LIN {X 0,Y 236.637,Z 407.423,A -85,B 0,C 180,E1 -20816.053,E2 -20816.053} C_VEL
LIN {X 0,Y 232.607,Z 398.672,A -85,B 0,C 180,E1 -20818.068,E2 -20818.068} C_VEL
LIN {X 0,Y 229.513,Z 389.934,A -85,B 0,C 180,E1 -20819.777,E2 -20819.777} C_VEL
LIN {X 0,Y 225.786,Z 379.77,A -85,B 0,C 180,E1 -20821.562,E2 -20821.562} C_VEL
LIN {X 0,Y 220.741,Z 368.882,A -85,B 0,C 180,E1 -20823.411,E2 -20823.411} C_VEL
LIN {X 0,Y 216.833,Z 361.674,A -85,B 0,C 180,E1 -20824.638,E2 -20824.638} C_VEL
LIN {X 0,Y 215.315,Z 358.971,A -85,B 0,C 180,E1 -20825.078,E2 -20825.078} C_VEL
LIN {X 0,Y 213.899,Z 356.173,A -85,B 0,C 180,E1 -20825.487,E2 -20825.487} C_VEL
LIN {X 0,Y 213.743,Z 355.361,A -85,B 0,C 180,E1 -20825.592,E2 -20825.592} C_VEL
LIN {X 0,Y 213.776,Z 355.356,A -85,B 0,C 180,E1 -20828.655,E2 -20828.655} C_VEL
LIN {X 0,Y 213.806,Z 355.353,A -85,B 0,C 180,E1 -20833.686,E2 -20833.686} C_VEL
LIN {X 0,Y 213.809,Z 355.352,A -85,B 0,C 180,E1 -20836.349,E2 -20836.349} C_VEL
LIN {X 0,Y 213.792,Z 355.354,A -85,B 0,C 180,E1 -20839.119,E2 -20839.119} C_VEL
LIN {X 0,Y 213.752,Z 355.359,A -85,B 0,C 180,E1 -20843.715,E2 -20843.715} C_VEL
LIN {X 0,Y 213.794,Z 355.352,A -85,B 0,C 180,E1 -20848.725,E2 -20848.725} C_VEL
LIN {X 0,Y 213.824,Z 355.349,A -85,B 0,C 180,E1 -20852.604,E2 -20852.604} C_VEL
LIN {X 0,Y 213.818,Z 355.35,A -85,B 0,C 180,E1 -20856.975,E2 -20856.975} C_VEL
LIN {X 0,Y 213.943,Z 355.336,A -85,B 0,C 180,E1 -20862.805,E2 -20862.805} C_VEL
LIN {X 0,Y 213.98,Z 355.328,A -85,B 0,C 180,E1 -20866.709,E2 -20866.709} C_VEL
LIN {X 0,Y 214.166,Z 355.301,A -85,B 0,C 180,E1 -20870.557,E2 -20870.557} C_VEL
LIN {X 0,Y 214.226,Z 355.299,A -85,B 0,C 180,E1 -20872.461,E2 -20872.461} C_VEL
LIN {X 0,Y 214.445,Z 355.244,A -85,B 0,C 180,E1 -20878.123,E2 -20878.123} C_VEL
LIN {X 0,Y 214.546,Z 355.244,A -85,B 0,C 180,E1 -20880.001,E2 -20880.001} C_VEL
LIN {X 0,Y 214.446,Z 355.269,A -85,B 0,C 180,E1 -20881.879,E2 -20881.879} C_VEL
LIN {X 0,Y 214.227,Z 355.3,A -85,B 0,C 180,E1 -20887.541,E2 -20887.541} C_VEL
LIN {X 0,Y 214.022,Z 355.327,A -85,B 0,C 180,E1 -20891.364,E2 -20891.364} C_VEL
LIN {X 0,Y 213.913,Z 355.341,A -85,B 0,C 180,E1 -20895.239,E2 -20895.239} C_VEL
LIN {X 0,Y 213.82,Z 355.351,A -85,B 0,C 180,E1 -20899.19,E2 -20899.19} C_VEL
LIN {X 0,Y 213.812,Z 355.353,A -85,B 0,C 180,E1 -20903.232,E2 -20903.232} C_VEL
LIN {X 0,Y 213.831,Z 355.54,A -85,B 0,C 180,E1 -20907.451,E2 -20907.451} C_VEL
LIN {X 0,Y 214.005,Z 357.167,A -85,B 0,C 180,E1 -20911.699,E2 -20911.699} C_VEL
LIN {X 0,Y 214.27,Z 359.11,A -85,B 0,C 180,E1 -20916.186,E2 -20916.186} C_VEL
LIN {X 0,Y 214.638,Z 361.528,A -85,B 0,C 180,E1 -20921.141,E2 -20921.141} C_VEL
LIN {X 0,Y 214.75,Z 363.018,A -85,B 0,C 180,E1 -20923.947,E2 -20923.947} C_VEL
LIN {X 0,Y 214.71,Z 364.508,A -85,B 0,C 180,E1 -20926.577,E2 -20926.577} C_VEL
LIN {X 0,Y 214.484,Z 365.996,A -85,B 0,C 180,E1 -20929.055,E2 -20929.055} C_VEL
LIN {X 0,Y 214.063,Z 367.842,A -85,B 0,C 180,E1 -20931.996,E2 -20931.996} C_VEL
LIN {X 0,Y 213.615,Z 369.611,A -85,B 0,C 180,E1 -20934.67,E2 -20934.67} C_VEL
LIN {X 0,Y 214.471,Z 372.783,A -85,B 0,C 180,E1 -20935.009,E2 -20935.009} C_VEL
LIN {X 0,Y 218.045,Z 383.16,A -85,B 0,C 180,E1 -20936.461,E2 -20936.461} C_VEL
LIN {X 0,Y 221.063,Z 395.512,A -85,B 0,C 180,E1 -20938.295,E2 -20938.295} C_VEL
LIN {X 0,Y 222.714,Z 405.325,A -85,B 0,C 180,E1 -20939.887,E2 -20939.887} C_VEL
LIN {X 0,Y 223.669,Z 414.982,A -85,B 0,C 180,E1 -20941.62,E2 -20941.62} C_VEL
LIN {X 0,Y 223.891,Z 424.106,A -85,B 0,C 180,E1 -20943.447,E2 -20943.447} C_VEL
LIN {X 0,Y 223.651,Z 428.588,A -85,B 0,C 180,E1 -20944.401,E2 -20944.401} C_VEL
LIN {X 0,Y 220.94,Z 438.166,A -85,B 0,C 180,E1 -20946.571,E2 -20946.571} C_VEL
LIN {X 0,Y 218.739,Z 445.725,A -85,B 0,C 180,E1 -20948.713,E2 -20948.713} C_VEL
LIN {X 0,Y 216.763,Z 452.535,A -85,B 0,C 180,E1 -20951.081,E2 -20951.081} C_VEL
LIN {X 0,Y 215.226,Z 457.725,A -85,B 0,C 180,E1 -20953.259,E2 -20953.259} C_VEL
LIN {X 0,Y 213.717,Z 460.581,A -85,B 0,C 180,E1 -20954.599,E2 -20954.599} C_VEL
LIN {X 0,Y 209.734,Z 464.564,A -85,B 0,C 180,E1 -20956.799,E2 -20956.799} C_VEL
LIN {X 0,Y 206.003,Z 467.926,A -85,B 0,C 180,E1 -20959.155,E2 -20959.155} C_VEL
LIN {X 0,Y 204.917,Z 469.562,A -85,B 0,C 180,E1 -20960.709,E2 -20960.709} C_VEL
LIN {X 0,Y 204.405,Z 472.228,A -85,B 0,C 180,E1 -20964.08,E2 -20964.08} C_VEL
LIN {X 0,Y 204.339,Z 473.292,A -85,B 0,C 180,E1 -20966.056,E2 -20966.056} C_VEL
LIN {X 0,Y 204.335,Z 473.885,A -85,B 0,C 180,E1 -20968.029,E2 -20968.029} C_VEL
LIN {X 0,Y 204.443,Z 474.044,A -85,B 0,C 180,E1 -20970,E2 -20970} C_VEL
LIN {X 0,Y 204.334,Z 473.885,A -85,B 0,C 180,E1 -20971.971,E2 -20971.971} C_VEL
LIN {X 0,Y 204.299,Z 473.291,A -85,B 0,C 180,E1 -20973.945,E2 -20973.945} C_VEL
LIN {X 0,Y 204.643,Z 470.836,A -85,B 0,C 180,E1 -20977.896,E2 -20977.896} C_VEL
LIN {X 0,Y 205.316,Z 467.882,A -85,B 0,C 180,E1 -20980.852,E2 -20980.852} C_VEL
LIN {X 0,Y 206.328,Z 463.887,A -85,B 0,C 180,E1 -20983.794,E2 -20983.794} C_VEL
LIN {X 0,Y 207.985,Z 458.757,A -85,B 0,C 180,E1 -20986.692,E2 -20986.692} C_VEL
LIN {X 0,Y 209.651,Z 453.494,A -85,B 0,C 180,E1 -20989.077,E2 -20989.077} C_VEL
LIN {X 0,Y 211.297,Z 448.555,A -85,B 0,C 180,E1 -20990.95,E2 -20990.95} C_VEL
LIN {X 0,Y 212.934,Z 442.852,A -85,B 0,C 180,E1 -20992.818,E2 -20992.818} C_VEL
LIN {X 0,Y 215.477,Z 434.299,A -85,B 0,C 180,E1 -20995.088,E2 -20995.088} C_VEL
LIN {X 0,Y 217.129,Z 428.388,A -85,B 0,C 180,E1 -20996.427,E2 -20996.427} C_VEL
LIN {X 0,Y 217.265,Z 418.838,A -85,B 0,C 180,E1 -20998.508,E2 -20998.508} C_VEL
LIN {X 0,Y 216.618,Z 409.561,A -85,B 0,C 180,E1 -21000.324,E2 -21000.324} C_VEL
LIN {X 0,Y 215.169,Z 399.419,A -85,B 0,C 180,E1 -21002.119,E2 -21002.119} C_VEL
LIN {X 0,Y 213.245,Z 390.302,A -85,B 0,C 180,E1 -21003.61,E2 -21003.61} C_VEL
LIN {X 0,Y 210.499,Z 380.51,A -85,B 0,C 180,E1 -21005.113,E2 -21005.113} C_VEL
LIN {X 0,Y 207.569,Z 372.479,A -85,B 0,C 180,E1 -21006.34,E2 -21006.34} C_VEL
LIN {X 0,Y 206.759,Z 369.447,A -85,B 0,C 180,E1 -21006.724,E2 -21006.724} C_VEL
LIN {X 0,Y 207.256,Z 367.276,A -85,B 0,C 180,E1 -21010.112,E2 -21010.112} C_VEL
LIN {X 0,Y 207.547,Z 365.774,A -85,B 0,C 180,E1 -21012.628,E2 -21012.628} C_VEL
LIN {X 0,Y 207.694,Z 364.302,A -85,B 0,C 180,E1 -21015.284,E2 -21015.284} C_VEL
LIN {X 0,Y 207.502,Z 361.92,A -85,B 0,C 180,E1 -21019.944,E2 -21019.944} C_VEL
LIN {X 0,Y 207.201,Z 359.698,A -85,B 0,C 180,E1 -21024.786,E2 -21024.786} C_VEL
LIN {X 0,Y 206.933,Z 357.824,A -85,B 0,C 180,E1 -21029.372,E2 -21029.372} C_VEL
LIN {X 0,Y 206.733,Z 356.236,A -85,B 0,C 180,E1 -21033.771,E2 -21033.771} C_VEL
LIN {X 0,Y 206.737,Z 356.236,A -85,B 0,C 180,E1 -21038.04,E2 -21038.04} C_VEL
LIN {X 0,Y 206.869,Z 356.218,A -85,B 0,C 180,E1 -21042.195,E2 -21042.195} C_VEL
LIN {X 0,Y 206.886,Z 356.214,A -85,B 0,C 180,E1 -21046.243,E2 -21046.243} C_VEL
LIN {X 0,Y 207.106,Z 356.186,A -85,B 0,C 180,E1 -21050.23,E2 -21050.23} C_VEL
LIN {X 0,Y 207.168,Z 356.179,A -85,B 0,C 180,E1 -21052.2,E2 -21052.2} C_VEL
LIN {X 0,Y 207.382,Z 356.149,A -85,B 0,C 180,E1 -21058.057,E2 -21058.057} C_VEL
LIN {X 0,Y 207.512,Z 356.118,A -85,B 0,C 180,E1 -21059.999,E2 -21059.999} C_VEL
LIN {X 0,Y 207.382,Z 356.122,A -85,B 0,C 180,E1 -21061.941,E2 -21061.941} C_VEL
LIN {X 0,Y 207.167,Z 356.178,A -85,B 0,C 180,E1 -21067.798,E2 -21067.798} C_VEL
LIN {X 0,Y 206.981,Z 356.202,A -85,B 0,C 180,E1 -21071.754,E2 -21071.754} C_VEL
LIN {X 0,Y 206.866,Z 356.213,A -85,B 0,C 180,E1 -21075.77,E2 -21075.77} C_VEL
LIN {X 0,Y 206.762,Z 356.222,A -85,B 0,C 180,E1 -21079.87,E2 -21079.87} C_VEL
LIN {X 0,Y 206.745,Z 356.228,A -85,B 0,C 180,E1 -21084.073,E2 -21084.073} C_VEL
LIN {X 0,Y 206.742,Z 356.232,A -85,B 0,C 180,E1 -21088.418,E2 -21088.418} C_VEL
LIN {X 0,Y 206.707,Z 356.235,A -85,B 0,C 180,E1 -21092.955,E2 -21092.955} C_VEL
LIN {X 0,Y 206.723,Z 356.235,A -85,B 0,C 180,E1 -21097.729,E2 -21097.729} C_VEL
LIN {X 0,Y 206.721,Z 356.235,A -85,B 0,C 180,E1 -21101.588,E2 -21101.588} C_VEL
LIN {X 0,Y 206.715,Z 356.234,A -85,B 0,C 180,E1 -21105.557,E2 -21105.557} C_VEL
LIN {X 0,Y 206.717,Z 356.235,A -85,B 0,C 180,E1 -21109.762,E2 -21109.762} C_VEL
LIN {X 0,Y 206.724,Z 356.235,A -85,B 0,C 180,E1 -21113.053,E2 -21113.053} C_VEL
LIN {X 0,Y 207.763,Z 359.167,A -85,B 0,C 180,E1 -21113.467,E2 -21113.467} C_VEL
LIN {X 0,Y 209.141,Z 361.156,A -85,B 0,C 180,E1 -21113.859,E2 -21113.859} C_VEL
LIN {X 0,Y 214.594,Z 371.285,A -85,B 0,C 180,E1 -21115.68,E2 -21115.68} C_VEL
LIN {X 0,Y 219.935,Z 383.191,A -85,B 0,C 180,E1 -21117.855,E2 -21117.855} C_VEL
LIN {X 0,Y 223.964,Z 394.74,A -85,B 0,C 180,E1 -21120.075,E2 -21120.075} C_VEL
LIN {X 0,Y 226.905,Z 403.215,A -85,B 0,C 180,E1 -21121.899,E2 -21121.899} C_VEL
LIN {X 0,Y 230.392,Z 410.806,A -85,B 0,C 180,E1 -21123.814,E2 -21123.814} C_VEL
LIN {X 0,Y 235.845,Z 419.628,A -85,B 0,C 180,E1 -21126.391,E2 -21126.391} C_VEL
LIN {X 0,Y 242.561,Z 427.895,A -85,B 0,C 180,E1 -21129.18,E2 -21129.18} C_VEL
LIN {X 0,Y 250.879,Z 435.889,A -85,B 0,C 180,E1 -21132.259,E2 -21132.259} C_VEL
LIN {X 0,Y 258.448,Z 441.903,A -85,B 0,C 180,E1 -21134.867,E2 -21134.867} C_VEL
LIN {X 0,Y 267.451,Z 447.962,A -85,B 0,C 180,E1 -21137.865,E2 -21137.865} C_VEL
LIN {X 0,Y 274.648,Z 452.392,A -85,B 0,C 180,E1 -21140.426,E2 -21140.426} C_VEL
LIN {X 0,Y 280.647,Z 455.777,A -85,B 0,C 180,E1 -21142.807,E2 -21142.807} C_VEL
LIN {X 0,Y 283.645,Z 457.491,A -85,B 0,C 180,E1 -21144.312,E2 -21144.312} C_VEL
LIN {X 0,Y 285.802,Z 458.811,A -85,B 0,C 180,E1 -21145.769,E2 -21145.769} C_VEL
LIN {X 0,Y 288.397,Z 459.95,A -85,B 0,C 180,E1 -21147.597,E2 -21147.597} C_VEL
LIN {X 0,Y 289.483,Z 460.298,A -85,B 0,C 180,E1 -21148.609,E2 -21148.609} C_VEL
LIN {X 0,Y 290.505,Z 460.469,A -85,B 0,C 180,E1 -21150,E2 -21150} C_VEL
LIN {X 0,Y 289.451,Z 460.299,A -85,B 0,C 180,E1 -21151.391,E2 -21151.391} C_VEL
LIN {X 0,Y 287.782,Z 459.753,A -85,B 0,C 180,E1 -21152.8,E2 -21152.8} C_VEL
LIN {X 0,Y 285.767,Z 458.812,A -85,B 0,C 180,E1 -21154.231,E2 -21154.231} C_VEL
LIN {X 0,Y 282.769,Z 456.952,A -85,B 0,C 180,E1 -21156.199,E2 -21156.199} C_VEL
LIN {X 0,Y 280.618,Z 455.778,A -85,B 0,C 180,E1 -21157.194,E2 -21157.194} C_VEL
LIN {X 0,Y 274.681,Z 452.391,A -85,B 0,C 180,E1 -21159.573,E2 -21159.573} C_VEL
LIN {X 0,Y 267.469,Z 447.961,A -85,B 0,C 180,E1 -21162.134,E2 -21162.134} C_VEL
LIN {X 0,Y 258.46,Z 441.872,A -85,B 0,C 180,E1 -21165.143,E2 -21165.143} C_VEL
LIN {X 0,Y 250.162,Z 435.246,A -85,B 0,C 180,E1 -21168.001,E2 -21168.001} C_VEL
LIN {X 0,Y 242.538,Z 427.896,A -85,B 0,C 180,E1 -21170.822,E2 -21170.822} C_VEL
LIN {X 0,Y 235.837,Z 419.654,A -85,B 0,C 180,E1 -21173.604,E2 -21173.604} C_VEL
LIN {X 0,Y 230.413,Z 410.784,A -85,B 0,C 180,E1 -21176.188,E2 -21176.188} C_VEL
LIN {X 0,Y 226.497,Z 402.035,A -85,B 0,C 180,E1 -21178.37,E2 -21178.37} C_VEL
LIN {X 0,Y 222.706,Z 390.823,A -85,B 0,C 180,E1 -21180.693,E2 -21180.693} C_VEL
LIN {X 0,Y 219.275,Z 381.514,A -85,B 0,C 180,E1 -21182.446,E2 -21182.446} C_VEL
LIN {X 0,Y 214.031,Z 370.166,A -85,B 0,C 180,E1 -21184.516,E2 -21184.516} C_VEL
LIN {X 0,Y 208.531,Z 360.174,A -85,B 0,C 180,E1 -21186.339,E2 -21186.339} C_VEL
LIN {X 0,Y 207.1,Z 357.827,A -85,B 0,C 180,E1 -21186.767,E2 -21186.767} C_VEL
LIN {X 0,Y 206.708,Z 356.237,A -85,B 0,C 180,E1 -21186.941,E2 -21186.941} C_VEL
LIN {X 0,Y 206.716,Z 356.236,A -85,B 0,C 180,E1 -21191.588,E2 -21191.588} C_VEL
LIN {X 0,Y 206.715,Z 356.235,A -85,B 0,C 180,E1 -21195.558,E2 -21195.558} C_VEL
LIN {X 0,Y 206.722,Z 356.234,A -85,B 0,C 180,E1 -21199.765,E2 -21199.765} C_VEL
LIN {X 0,Y 206.723,Z 356.235,A -85,B 0,C 180,E1 -21202.271,E2 -21202.271} C_VEL
LIN {X 0,Y 206.707,Z 356.235,A -85,B 0,C 180,E1 -21207.045,E2 -21207.045} C_VEL
LIN {X 0,Y 206.765,Z 356.229,A -85,B 0,C 180,E1 -21212.097,E2 -21212.097} C_VEL
LIN {X 0,Y 206.753,Z 356.229,A -85,B 0,C 180,E1 -21216.605,E2 -21216.605} C_VEL
LIN {X 0,Y 206.872,Z 356.215,A -85,B 0,C 180,E1 -21222.198,E2 -21222.198} C_VEL
LIN {X 0,Y 206.913,Z 356.207,A -85,B 0,C 180,E1 -21226.247,E2 -21226.247} C_VEL
LIN {X 0,Y 207.105,Z 356.18,A -85,B 0,C 180,E1 -21230.232,E2 -21230.232} C_VEL
LIN {X 0,Y 207.167,Z 356.178,A -85,B 0,C 180,E1 -21232.202,E2 -21232.202} C_VEL
LIN {X 0,Y 207.382,Z 356.122,A -85,B 0,C 180,E1 -21238.059,E2 -21238.059} C_VEL
LIN {X 0,Y 207.512,Z 356.118,A -85,B 0,C 180,E1 -21240.001,E2 -21240.001} C_VEL
LIN {X 0,Y 207.382,Z 356.149,A -85,B 0,C 180,E1 -21241.943,E2 -21241.943} C_VEL
LIN {X 0,Y 207.168,Z 356.179,A -85,B 0,C 180,E1 -21247.8,E2 -21247.8} C_VEL
LIN {X 0,Y 206.941,Z 356.209,A -85,B 0,C 180,E1 -21251.758,E2 -21251.758} C_VEL
LIN {X 0,Y 206.846,Z 356.221,A -85,B 0,C 180,E1 -21255.773,E2 -21255.773} C_VEL
LIN {X 0,Y 206.858,Z 356.22,A -85,B 0,C 180,E1 -21257.955,E2 -21257.955} C_VEL
LIN {X 0,Y 206.755,Z 356.233,A -85,B 0,C 180,E1 -21263.397,E2 -21263.397} C_VEL
LIN {X 0,Y 206.732,Z 356.236,A -85,B 0,C 180,E1 -21266.229,E2 -21266.229} C_VEL
LIN {X 0,Y 206.933,Z 357.826,A -85,B 0,C 180,E1 -21270.628,E2 -21270.628} C_VEL
LIN {X 0,Y 207.209,Z 359.819,A -85,B 0,C 180,E1 -21275.51,E2 -21275.51} C_VEL
LIN {X 0,Y 207.507,Z 361.919,A -85,B 0,C 180,E1 -21280.055,E2 -21280.055} C_VEL
LIN {X 0,Y 207.633,Z 363.198,A -85,B 0,C 180,E1 -21282.608,E2 -21282.608} C_VEL
LIN {X 0,Y 207.679,Z 364.638,A -85,B 0,C 180,E1 -21285.29,E2 -21285.29} C_VEL
LIN {X 0,Y 207.479,Z 366.287,A -85,B 0,C 180,E1 -21288.179,E2 -21288.179} C_VEL
LIN {X 0,Y 206.907,Z 368.745,A -85,B 0,C 180,E1 -21292.309,E2 -21292.309} C_VEL
LIN {X 0,Y 206.749,Z 369.396,A -85,B 0,C 180,E1 -21293.278,E2 -21293.278} C_VEL
LIN {X 0,Y 207.674,Z 372.711,A -85,B 0,C 180,E1 -21293.696,E2 -21293.696} C_VEL
LIN {X 0,Y 209.982,Z 379.098,A -85,B 0,C 180,E1 -21294.671,E2 -21294.671} C_VEL
LIN {X 0,Y 212.326,Z 386.827,A -85,B 0,C 180,E1 -21295.845,E2 -21295.845} C_VEL
LIN {X 0,Y 214.591,Z 396.436,A -85,B 0,C 180,E1 -21297.377,E2 -21297.377} C_VEL
LIN {X 0,Y 216.196,Z 406.3,A -85,B 0,C 180,E1 -21299.076,E2 -21299.076} C_VEL
LIN {X 0,Y 217.01,Z 414.175,A -85,B 0,C 180,E1 -21300.549,E2 -21300.549} C_VEL
LIN {X 0,Y 217.308,Z 422.163,A -85,B 0,C 180,E1 -21302.179,E2 -21302.179} C_VEL
LIN {X 0,Y 216.962,Z 429.481,A -85,B 0,C 180,E1 -21303.81,E2 -21303.81} C_VEL
LIN {X 0,Y 214.432,Z 437.97,A -85,B 0,C 180,E1 -21305.815,E2 -21305.815} C_VEL
LIN {X 0,Y 211.879,Z 446.215,A -85,B 0,C 180,E1 -21308.244,E2 -21308.244} C_VEL
LIN {X 0,Y 210.044,Z 452.339,A -85,B 0,C 180,E1 -21310.452,E2 -21310.452} C_VEL
LIN {X 0,Y 208.278,Z 457.897,A -85,B 0,C 180,E1 -21312.879,E2 -21312.879} C_VEL
LIN {X 0,Y 206.823,Z 462.333,A -85,B 0,C 180,E1 -21315.235,E2 -21315.235} C_VEL
LIN {X 0,Y 205.608,Z 466.663,A -85,B 0,C 180,E1 -21318.165,E2 -21318.165} C_VEL
LIN {X 0,Y 204.917,Z 469.562,A -85,B 0,C 180,E1 -21320.709,E2 -21320.709} C_VEL
LIN {X 0,Y 203.933,Z 471.027,A -85,B 0,C 180,E1 -21322.298,E2 -21322.298} C_VEL
LIN {X 0,Y 200.776,Z 472.689,A -85,B 0,C 180,E1 -21324.921,E2 -21324.921} C_VEL
LIN {X 0,Y 198.305,Z 473.463,A -85,B 0,C 180,E1 -21327.089,E2 -21327.089} C_VEL
LIN {X 0,Y 197.33,Z 473.846,A -85,B 0,C 180,E1 -21328.787,E2 -21328.787} C_VEL
LIN {X 0,Y 197.286,Z 473.799,A -85,B 0,C 180,E1 -21329.363,E2 -21329.363} C_VEL
LIN {X 0,Y 197.24,Z 473.69,A -85,B 0,C 180,E1 -21332.042,E2 -21332.042} C_VEL
LIN {X 0,Y 197.21,Z 473.095,A -85,B 0,C 180,E1 -21334.087,E2 -21334.087} C_VEL
LIN {X 0,Y 197.593,Z 470.64,A -85,B 0,C 180,E1 -21338.179,E2 -21338.179} C_VEL
LIN {X 0,Y 198.302,Z 467.685,A -85,B 0,C 180,E1 -21341.24,E2 -21341.24} C_VEL
LIN {X 0,Y 199.401,Z 463.69,A -85,B 0,C 180,E1 -21344.283,E2 -21344.283} C_VEL
LIN {X 0,Y 201.166,Z 458.561,A -85,B 0,C 180,E1 -21347.275,E2 -21347.275} C_VEL
LIN {X 0,Y 202.931,Z 453.298,A -85,B 0,C 180,E1 -21349.735,E2 -21349.735} C_VEL
LIN {X 0,Y 204.622,Z 448.36,A -85,B 0,C 180,E1 -21351.666,E2 -21351.666} C_VEL
LIN {X 0,Y 206.386,Z 442.656,A -85,B 0,C 180,E1 -21353.585,E2 -21353.585} C_VEL
LIN {X 0,Y 209.045,Z 434.102,A -85,B 0,C 180,E1 -21355.916,E2 -21355.916} C_VEL
LIN {X 0,Y 210.473,Z 429.28,A -85,B 0,C 180,E1 -21357.062,E2 -21357.062} C_VEL
LIN {X 0,Y 210.656,Z 418.629,A -85,B 0,C 180,E1 -21359.489,E2 -21359.489} C_VEL
LIN {X 0,Y 210.109,Z 410.083,A -85,B 0,C 180,E1 -21361.243,E2 -21361.243} C_VEL
LIN {X 0,Y 208.677,Z 400.01,A -85,B 0,C 180,E1 -21363.131,E2 -21363.131} C_VEL
LIN {X 0,Y 206.655,Z 390.343,A -85,B 0,C 180,E1 -21364.803,E2 -21364.803} C_VEL
LIN {X 0,Y 203.664,Z 380.15,A -85,B 0,C 180,E1 -21366.487,E2 -21366.487} C_VEL
LIN {X 0,Y 200.915,Z 372.676,A -85,B 0,C 180,E1 -21367.72,E2 -21367.72} C_VEL
LIN {X 0,Y 199.941,Z 369.241,A -85,B 0,C 180,E1 -21368.184,E2 -21368.184} C_VEL
LIN {X 0,Y 200.495,Z 366.607,A -85,B 0,C 180,E1 -21372.597,E2 -21372.597} C_VEL
LIN {X 0,Y 200.631,Z 365.04,A -85,B 0,C 180,E1 -21375.524,E2 -21375.524} C_VEL
LIN {X 0,Y 200.567,Z 363.667,A -85,B 0,C 180,E1 -21378.257,E2 -21378.257} C_VEL
LIN {X 0,Y 200.39,Z 362.457,A -85,B 0,C 180,E1 -21380.854,E2 -21380.854} C_VEL
LIN {X 0,Y 200.081,Z 360.307,A -85,B 0,C 180,E1 -21385.804,E2 -21385.804} C_VEL
LIN {X 0,Y 199.821,Z 358.473,A -85,B 0,C 180,E1 -21390.5,E2 -21390.5} C_VEL
LIN {X 0,Y 199.666,Z 357.116,A -85,B 0,C 180,E1 -21395.014,E2 -21395.014} C_VEL
LIN {X 0,Y 199.675,Z 357.116,A -85,B 0,C 180,E1 -21399.391,E2 -21399.391} C_VEL
LIN {X 0,Y 199.79,Z 357.1,A -85,B 0,C 180,E1 -21403.654,E2 -21403.654} C_VEL
LIN {X 0,Y 200.037,Z 357.069,A -85,B 0,C 180,E1 -21409.652,E2 -21409.652} C_VEL
LIN {X 0,Y 200.112,Z 357.059,A -85,B 0,C 180,E1 -21411.923,E2 -21411.923} C_VEL
LIN {X 0,Y 200.322,Z 357.028,A -85,B 0,C 180,E1 -21417.988,E2 -21417.988} C_VEL
LIN {X 0,Y 200.476,Z 356.993,A -85,B 0,C 180,E1 -21419.999,E2 -21419.999} C_VEL
LIN {X 0,Y 200.03,Z 357.053,A -85,B 0,C 180,E1 -21424.028,E2 -21424.028} C_VEL
LIN {X 0,Y 200.11,Z 357.057,A -85,B 0,C 180,E1 -21428.075,E2 -21428.075} C_VEL
LIN {X 0,Y 199.913,Z 357.083,A -85,B 0,C 180,E1 -21432.176,E2 -21432.176} C_VEL
LIN {X 0,Y 199.804,Z 357.094,A -85,B 0,C 180,E1 -21436.342,E2 -21436.342} C_VEL
LIN {X 0,Y 199.681,Z 357.106,A -85,B 0,C 180,E1 -21440.606,E2 -21440.606} C_VEL
LIN {X 0,Y 199.663,Z 357.107,A -85,B 0,C 180,E1 -21444.984,E2 -21444.984} C_VEL
LIN {X 0,Y 199.673,Z 357.112,A -85,B 0,C 180,E1 -21449.521,E2 -21449.521} C_VEL
LIN {X 0,Y 199.663,Z 357.116,A -85,B 0,C 180,E1 -21452.352,E2 -21452.352} C_VEL
LIN {X 0,Y 199.651,Z 357.116,A -85,B 0,C 180,E1 -21456.756,E2 -21456.756} C_VEL
LIN {X 0,Y 199.676,Z 357.112,A -85,B 0,C 180,E1 -21459.311,E2 -21459.311} C_VEL
LIN {X 0,Y 199.66,Z 357.114,A -85,B 0,C 180,E1 -21462.337,E2 -21462.337} C_VEL
LIN {X 0,Y 199.663,Z 357.112,A -85,B 0,C 180,E1 -21465.253,E2 -21465.253} C_VEL
LIN {X 0,Y 199.659,Z 357.115,A -85,B 0,C 180,E1 -21468.026,E2 -21468.026} C_VEL
LIN {X 0,Y 199.703,Z 357.11,A -85,B 0,C 180,E1 -21471.554,E2 -21471.554} C_VEL
LIN {X 0,Y 200.771,Z 360.098,A -85,B 0,C 180,E1 -21472.015,E2 -21472.015} C_VEL
LIN {X 0,Y 202.263,Z 362.257,A -85,B 0,C 180,E1 -21472.471,E2 -21472.471} C_VEL
LIN {X 0,Y 208.682,Z 374.094,A -85,B 0,C 180,E1 -21474.805,E2 -21474.805} C_VEL
LIN {X 0,Y 213.987,Z 386.324,A -85,B 0,C 180,E1 -21477.243,E2 -21477.243} C_VEL
LIN {X 0,Y 217.48,Z 396.565,A -85,B 0,C 180,E1 -21479.358,E2 -21479.358} C_VEL
LIN {X 0,Y 219.941,Z 404.442,A -85,B 0,C 180,E1 -21481.122,E2 -21481.122} C_VEL
LIN {X 0,Y 223.105,Z 412.162,A -85,B 0,C 180,E1 -21483.127,E2 -21483.127} C_VEL
LIN {X 0,Y 228.164,Z 420.867,A -85,B 0,C 180,E1 -21485.798,E2 -21485.798} C_VEL
LIN {X 0,Y 234.108,Z 428.619,A -85,B 0,C 180,E1 -21488.53,E2 -21488.53} C_VEL
LIN {X 0,Y 240.871,Z 435.51,A -85,B 0,C 180,E1 -21491.28,E2 -21491.28} C_VEL
LIN {X 0,Y 248.484,Z 441.722,A -85,B 0,C 180,E1 -21494.075,E2 -21494.075} C_VEL
LIN {X 0,Y 255.89,Z 446.803,A -85,B 0,C 180,E1 -21496.65,E2 -21496.65} C_VEL
LIN {X 0,Y 263.403,Z 451.269,A -85,B 0,C 180,E1 -21499.236,E2 -21499.236} C_VEL
LIN {X 0,Y 269.931,Z 454.79,A -85,B 0,C 180,E1 -21501.635,E2 -21501.635} C_VEL
LIN {X 0,Y 275.584,Z 457.589,A -85,B 0,C 180,E1 -21504.026,E2 -21504.026} C_VEL
LIN {X 0,Y 278.245,Z 459.019,A -85,B 0,C 180,E1 -21505.654,E2 -21505.654} C_VEL
LIN {X 0,Y 281.323,Z 460.246,A -85,B 0,C 180,E1 -21507.798,E2 -21507.798} C_VEL
LIN {X 0,Y 282.195,Z 460.498,A -85,B 0,C 180,E1 -21508.573,E2 -21508.573} C_VEL
LIN {X 0,Y 283.336,Z 460.663,A -85,B 0,C 180,E1 -21510,E2 -21510} C_VEL
LIN {X 0,Y 282.158,Z 460.5,A -85,B 0,C 180,E1 -21511.427,E2 -21511.427} C_VEL
LIN {X 0,Y 280.293,Z 459.961,A -85,B 0,C 180,E1 -21512.874,E2 -21512.874} C_VEL
LIN {X 0,Y 278.223,Z 459.019,A -85,B 0,C 180,E1 -21514.346,E2 -21514.346} C_VEL
LIN {X 0,Y 275.584,Z 457.589,A -85,B 0,C 180,E1 -21515.974,E2 -21515.974} C_VEL
LIN {X 0,Y 269.933,Z 454.787,A -85,B 0,C 180,E1 -21518.368,E2 -21518.368} C_VEL
LIN {X 0,Y 264.389,Z 451.84,A -85,B 0,C 180,E1 -21520.417,E2 -21520.417} C_VEL
LIN {X 0,Y 258.176,Z 448.225,A -85,B 0,C 180,E1 -21522.578,E2 -21522.578} C_VEL
LIN {X 0,Y 250.51,Z 443.219,A -85,B 0,C 180,E1 -21525.209,E2 -21525.209} C_VEL
LIN {X 0,Y 242.177,Z 436.691,A -85,B 0,C 180,E1 -21528.222,E2 -21528.222} C_VEL
LIN {X 0,Y 235.17,Z 429.821,A -85,B 0,C 180,E1 -21531.015,E2 -21531.015} C_VEL
LIN {X 0,Y 229.703,Z 423.161,A -85,B 0,C 180,E1 -21533.437,E2 -21533.437} C_VEL
LIN {X 0,Y 224.75,Z 415.246,A -85,B 0,C 180,E1 -21535.962,E2 -21535.962} C_VEL
LIN {X 0,Y 221.163,Z 407.631,A -85,B 0,C 180,E1 -21538.078,E2 -21538.078} C_VEL
LIN {X 0,Y 217.831,Z 398.026,A -85,B 0,C 180,E1 -21540.343,E2 -21540.343} C_VEL
LIN {X 0,Y 214.997,Z 388.99,A -85,B 0,C 180,E1 -21542.209,E2 -21542.209} C_VEL
LIN {X 0,Y 211.104,Z 379.389,A -85,B 0,C 180,E1 -21544.137,E2 -21544.137} C_VEL
LIN {X 0,Y 206.394,Z 369.786,A -85,B 0,C 180,E1 -21546.041,E2 -21546.041} C_VEL
LIN {X 0,Y 201.443,Z 360.977,A -85,B 0,C 180,E1 -21547.801,E2 -21547.801} C_VEL
LIN {X 0,Y 199.989,Z 358.348,A -85,B 0,C 180,E1 -21548.29,E2 -21548.29} C_VEL
LIN {X 0,Y 199.704,Z 357.11,A -85,B 0,C 180,E1 -21548.459,E2 -21548.459} C_VEL
LIN {X 0,Y 199.657,Z 357.114,A -85,B 0,C 180,E1 -21552.338,E2 -21552.338} C_VEL
LIN {X 0,Y 199.663,Z 357.112,A -85,B 0,C 180,E1 -21555.254,E2 -21555.254} C_VEL
LIN {X 0,Y 199.664,Z 357.115,A -85,B 0,C 180,E1 -21558.028,E2 -21558.028} C_VEL
LIN {X 0,Y 199.678,Z 357.112,A -85,B 0,C 180,E1 -21560.744,E2 -21560.744} C_VEL
LIN {X 0,Y 199.633,Z 357.118,A -85,B 0,C 180,E1 -21565.719,E2 -21565.719} C_VEL
LIN {X 0,Y 199.702,Z 357.109,A -85,B 0,C 180,E1 -21568.139,E2 -21568.139} C_VEL
LIN {X 0,Y 199.685,Z 357.111,A -85,B 0,C 180,E1 -21572.773,E2 -21572.773} C_VEL
LIN {X 0,Y 199.713,Z 357.108,A -85,B 0,C 180,E1 -21577.227,E2 -21577.227} C_VEL
LIN {X 0,Y 199.795,Z 357.098,A -85,B 0,C 180,E1 -21581.759,E2 -21581.759} C_VEL
LIN {X 0,Y 199.847,Z 357.086,A -85,B 0,C 180,E1 -21585.75,E2 -21585.75} C_VEL
LIN {X 0,Y 200.07,Z 357.057,A -85,B 0,C 180,E1 -21589.885,E2 -21589.885} C_VEL
LIN {X 0,Y 200.034,Z 357.066,A -85,B 0,C 180,E1 -21593.951,E2 -21593.951} C_VEL
LIN {X 0,Y 200.321,Z 357.001,A -85,B 0,C 180,E1 -21597.991,E2 -21597.991} C_VEL
LIN {X 0,Y 200.476,Z 356.993,A -85,B 0,C 180,E1 -21600.001,E2 -21600.001} C_VEL
LIN {X 0,Y 200.031,Z 357.068,A -85,B 0,C 180,E1 -21604.031,E2 -21604.031} C_VEL
LIN {X 0,Y 200.112,Z 357.059,A -85,B 0,C 180,E1 -21608.077,E2 -21608.077} C_VEL
LIN {X 0,Y 200.037,Z 357.07,A -85,B 0,C 180,E1 -21610.348,E2 -21610.348} C_VEL
LIN {X 0,Y 199.79,Z 357.101,A -85,B 0,C 180,E1 -21616.346,E2 -21616.346} C_VEL
LIN {X 0,Y 199.675,Z 357.113,A -85,B 0,C 180,E1 -21620.609,E2 -21620.609} C_VEL
LIN {X 0,Y 199.666,Z 357.116,A -85,B 0,C 180,E1 -21624.986,E2 -21624.986} C_VEL
LIN {X 0,Y 199.82,Z 358.471,A -85,B 0,C 180,E1 -21629.5,E2 -21629.5} C_VEL
LIN {X 0,Y 200.083,Z 360.291,A -85,B 0,C 180,E1 -21634.196,E2 -21634.196} C_VEL
LIN {X 0,Y 200.426,Z 362.621,A -85,B 0,C 180,E1 -21639.517,E2 -21639.517} C_VEL
LIN {X 0,Y 200.588,Z 364.111,A -85,B 0,C 180,E1 -21642.627,E2 -21642.627} C_VEL
LIN {X 0,Y 200.611,Z 365.614,A -85,B 0,C 180,E1 -21645.52,E2 -21645.52} C_VEL
LIN {X 0,Y 200.401,Z 367.096,A -85,B 0,C 180,E1 -21648.216,E2 -21648.216} C_VEL
LIN {X 0,Y 199.93,Z 369.22,A -85,B 0,C 180,E1 -21651.838,E2 -21651.838} C_VEL
LIN {X 0,Y 200.79,Z 372.411,A -85,B 0,C 180,E1 -21652.234,E2 -21652.234} C_VEL
LIN {X 0,Y 201.852,Z 375.103,A -85,B 0,C 180,E1 -21652.687,E2 -21652.687} C_VEL
LIN {X 0,Y 204.99,Z 384.029,A -85,B 0,C 180,E1 -21654.144,E2 -21654.144} C_VEL
LIN {X 0,Y 207.904,Z 395.999,A -85,B 0,C 180,E1 -21656.159,E2 -21656.159} C_VEL
LIN {X 0,Y 209.612,Z 406.087,A -85,B 0,C 180,E1 -21657.992,E2 -21657.992} C_VEL
LIN {X 0,Y 210.458,Z 414.848,A -85,B 0,C 180,E1 -21659.716,E2 -21659.716} C_VEL
LIN {X 0,Y 210.704,Z 422.463,A -85,B 0,C 180,E1 -21661.348,E2 -21661.348} C_VEL
LIN {X 0,Y 210.3,Z 430.267,A -85,B 0,C 180,E1 -21663.182,E2 -21663.182} C_VEL
LIN {X 0,Y 207.403,Z 439.4,A -85,B 0,C 180,E1 -21665.474,E2 -21665.474} C_VEL
LIN {X 0,Y 204.985,Z 446.979,A -85,B 0,C 180,E1 -21667.843,E2 -21667.843} C_VEL
LIN {X 0,Y 203.358,Z 452.143,A -85,B 0,C 180,E1 -21669.782,E2 -21669.782} C_VEL
LIN {X 0,Y 201.863,Z 456.645,A -85,B 0,C 180,E1 -21671.739,E2 -21671.739} C_VEL
LIN {X 0,Y 199.925,Z 462.136,A -85,B 0,C 180,E1 -21674.713,E2 -21674.713} C_VEL
LIN {X 0,Y 198.627,Z 466.466,A -85,B 0,C 180,E1 -21677.743,E2 -21677.743} C_VEL
LIN {X 0,Y 197.834,Z 469.544,A -85,B 0,C 180,E1 -21680.578,E2 -21680.578} C_VEL
LIN {X 0,Y 197.344,Z 472.033,A -85,B 0,C 180,E1 -21683.867,E2 -21683.867} C_VEL
LIN {X 0,Y 197.248,Z 473.146,A -85,B 0,C 180,E1 -21686.085,E2 -21686.085} C_VEL
LIN {X 0,Y 197.286,Z 473.799,A -85,B 0,C 180,E1 -21689.363,E2 -21689.363} C_VEL
LIN {X 0,Y 196.68,Z 473.837,A -85,B 0,C 180,E1 -21691.063,E2 -21691.063} C_VEL
LIN {X 0,Y 195.087,Z 473.502,A -85,B 0,C 180,E1 -21692.733,E2 -21692.733} C_VEL
LIN {X 0,Y 191.395,Z 471.997,A -85,B 0,C 180,E1 -21696.095,E2 -21696.095} C_VEL
LIN {X 0,Y 190.52,Z 470.974,A -85,B 0,C 180,E1 -21697.842,E2 -21697.842} C_VEL
LIN {X 0,Y 190.534,Z 470.478,A -85,B 0,C 180,E1 -21698.432,E2 -21698.432} C_VEL
LIN {X 0,Y 191.31,Z 467.488,A -85,B 0,C 180,E1 -21701.657,E2 -21701.657} C_VEL
LIN {X 0,Y 192.49,Z 463.493,A -85,B 0,C 180,E1 -21704.808,E2 -21704.808} C_VEL
LIN {X 0,Y 194.372,Z 458.364,A -85,B 0,C 180,E1 -21707.899,E2 -21707.899} C_VEL
LIN {X 0,Y 196.248,Z 453.101,A -85,B 0,C 180,E1 -21710.436,E2 -21710.436} C_VEL
LIN {X 0,Y 198.02,Z 448.07,A -85,B 0,C 180,E1 -21712.464,E2 -21712.464} C_VEL
LIN {X 0,Y 200.362,Z 440.829,A -85,B 0,C 180,E1 -21714.892,E2 -21714.892} C_VEL
LIN {X 0,Y 202.67,Z 433.906,A -85,B 0,C 180,E1 -21716.795,E2 -21716.795} C_VEL
LIN {X 0,Y 203.921,Z 429.077,A -85,B 0,C 180,E1 -21718.007,E2 -21718.007} C_VEL
LIN {X 0,Y 204.14,Z 419.736,A -85,B 0,C 180,E1 -21720.253,E2 -21720.253} C_VEL
LIN {X 0,Y 203.448,Z 409.58,A -85,B 0,C 180,E1 -21722.439,E2 -21722.439} C_VEL
LIN {X 0,Y 202.2,Z 400.361,A -85,B 0,C 180,E1 -21724.253,E2 -21724.253} C_VEL
LIN {X 0,Y 200.087,Z 390.216,A -85,B 0,C 180,E1 -21726.11,E2 -21726.11} C_VEL
LIN {X 0,Y 196.96,Z 380.066,A -85,B 0,C 180,E1 -21727.93,E2 -21727.93} C_VEL
LIN {X 0,Y 194.246,Z 372.689,A -85,B 0,C 180,E1 -21729.238,E2 -21729.238} C_VEL
LIN {X 0,Y 193.192,Z 369.887,A -85,B 0,C 180,E1 -21729.678,E2 -21729.678} C_VEL
LIN {X 0,Y 193.082,Z 369.012,A -85,B 0,C 180,E1 -21729.817,E2 -21729.817} C_VEL
LIN {X 0,Y 193.488,Z 366.865,A -85,B 0,C 180,E1 -21733.64,E2 -21733.64} C_VEL
LIN {X 0,Y 193.546,Z 365.391,A -85,B 0,C 180,E1 -21736.571,E2 -21736.571} C_VEL
LIN {X 0,Y 193.426,Z 363.895,A -85,B 0,C 180,E1 -21739.731,E2 -21739.731} C_VEL
LIN {X 0,Y 193.123,Z 361.905,A -85,B 0,C 180,E1 -21744.389,E2 -21744.389} C_VEL
LIN {X 0,Y 193.017,Z 360.913,A -85,B 0,C 180,E1 -21746.894,E2 -21746.894} C_VEL
LIN {X 0,Y 192.778,Z 359.152,A -85,B 0,C 180,E1 -21751.709,E2 -21751.709} C_VEL
LIN {X 0,Y 192.648,Z 357.991,A -85,B 0,C 180,E1 -21755.786,E2 -21755.786} C_VEL
LIN {X 0,Y 192.731,Z 357.98,A -85,B 0,C 180,E1 -21761.459,E2 -21761.459} C_VEL
LIN {X 0,Y 192.753,Z 357.976,A -85,B 0,C 180,E1 -21765.212,E2 -21765.212} C_VEL
LIN {X 0,Y 192.982,Z 357.948,A -85,B 0,C 180,E1 -21769.507,E2 -21769.507} C_VEL
LIN {X 0,Y 193.062,Z 357.937,A -85,B 0,C 180,E1 -21771.626,E2 -21771.626} C_VEL
LIN {X 0,Y 193.264,Z 357.907,A -85,B 0,C 180,E1 -21777.915,E2 -21777.915} C_VEL
LIN {X 0,Y 193.441,Z 357.867,A -85,B 0,C 180,E1 -21779.999,E2 -21779.999} C_VEL
LIN {X 0,Y 192.976,Z 357.932,A -85,B 0,C 180,E1 -21784.176,E2 -21784.176} C_VEL
LIN {X 0,Y 193.061,Z 357.934,A -85,B 0,C 180,E1 -21788.372,E2 -21788.372} C_VEL
LIN {X 0,Y 192.852,Z 357.964,A -85,B 0,C 180,E1 -21792.629,E2 -21792.629} C_VEL
LIN {X 0,Y 192.756,Z 357.976,A -85,B 0,C 180,E1 -21796.958,E2 -21796.958} C_VEL
LIN {X 0,Y 192.616,Z 357.991,A -85,B 0,C 180,E1 -21801.398,E2 -21801.398} C_VEL
LIN {X 0,Y 192.646,Z 357.982,A -85,B 0,C 180,E1 -21804.212,E2 -21804.212} C_VEL
LIN {X 0,Y 192.648,Z 357.988,A -85,B 0,C 180,E1 -21808.891,E2 -21808.891} C_VEL
LIN {X 0,Y 192.599,Z 357.992,A -85,B 0,C 180,E1 -21813.184,E2 -21813.184} C_VEL
LIN {X 0,Y 192.598,Z 357.994,A -85,B 0,C 180,E1 -21818.339,E2 -21818.339} C_VEL
LIN {X 0,Y 192.602,Z 357.993,A -85,B 0,C 180,E1 -21823.131,E2 -21823.131} C_VEL
LIN {X 0,Y 192.6,Z 357.992,A -85,B 0,C 180,E1 -21826.868,E2 -21826.868} C_VEL
LIN {X 0,Y 192.613,Z 358.145,A -85,B 0,C 180,E1 -21829.951,E2 -21829.951} C_VEL
LIN {X 0,Y 193.785,Z 361.109,A -85,B 0,C 180,E1 -21830.432,E2 -21830.432} C_VEL
LIN {X 0,Y 195.234,Z 362.91,A -85,B 0,C 180,E1 -21830.896,E2 -21830.896} C_VEL
LIN {X 0,Y 202.062,Z 375.535,A -85,B 0,C 180,E1 -21833.606,E2 -21833.606} C_VEL
LIN {X 0,Y 206.818,Z 386.325,A -85,B 0,C 180,E1 -21835.923,E2 -21835.923} C_VEL
LIN {X 0,Y 210.223,Z 395.904,A -85,B 0,C 180,E1 -21838.025,E2 -21838.025} C_VEL
LIN {X 0,Y 213.12,Z 405.865,A -85,B 0,C 180,E1 -21840.353,E2 -21840.353} C_VEL
LIN {X 0,Y 216.847,Z 415.481,A -85,B 0,C 180,E1 -21843.016,E2 -21843.016} C_VEL
LIN {X 0,Y 221.396,Z 423.405,A -85,B 0,C 180,E1 -21845.627,E2 -21845.627} C_VEL
LIN {X 0,Y 226.829,Z 430.674,A -85,B 0,C 180,E1 -21848.356,E2 -21848.356} C_VEL
LIN {X 0,Y 234.89,Z 438.63,A -85,B 0,C 180,E1 -21851.795,E2 -21851.795} C_VEL
LIN {X 0,Y 243.157,Z 444.905,A -85,B 0,C 180,E1 -21854.922,E2 -21854.922} C_VEL
LIN {X 0,Y 251.564,Z 450.07,A -85,B 0,C 180,E1 -21857.9,E2 -21857.9} C_VEL
LIN {X 0,Y 259.269,Z 454.117,A -85,B 0,C 180,E1 -21860.64,E2 -21860.64} C_VEL
LIN {X 0,Y 263.834,Z 456.245,A -85,B 0,C 180,E1 -21862.346,E2 -21862.346} C_VEL
LIN {X 0,Y 268.392,Z 458.226,A -85,B 0,C 180,E1 -21864.288,E2 -21864.288} C_VEL
LIN {X 0,Y 270.584,Z 459.229,A -85,B 0,C 180,E1 -21865.531,E2 -21865.531} C_VEL
LIN {X 0,Y 274.25,Z 460.539,A -85,B 0,C 180,E1 -21868.024,E2 -21868.024} C_VEL
LIN {X 0,Y 276.153,Z 460.858,A -85,B 0,C 180,E1 -21870,E2 -21870} C_VEL
LIN {X 0,Y 274.246,Z 460.549,A -85,B 0,C 180,E1 -21871.948,E2 -21871.948} C_VEL
LIN {X 0,Y 270.555,Z 459.229,A -85,B 0,C 180,E1 -21874.469,E2 -21874.469} C_VEL
LIN {X 0,Y 267.64,Z 457.937,A -85,B 0,C 180,E1 -21876.029,E2 -21876.029} C_VEL
LIN {X 0,Y 262.655,Z 455.716,A -85,B 0,C 180,E1 -21878.105,E2 -21878.105} C_VEL
LIN {X 0,Y 257.045,Z 452.993,A -85,B 0,C 180,E1 -21880.173,E2 -21880.173} C_VEL
LIN {X 0,Y 248.788,Z 448.493,A -85,B 0,C 180,E1 -21883.061,E2 -21883.061} C_VEL
LIN {X 0,Y 241.073,Z 443.443,A -85,B 0,C 180,E1 -21885.84,E2 -21885.84} C_VEL
LIN {X 0,Y 233.69,Z 437.587,A -85,B 0,C 180,E1 -21888.685,E2 -21888.685} C_VEL
LIN {X 0,Y 226.338,Z 430.075,A -85,B 0,C 180,E1 -21891.877,E2 -21891.877} C_VEL
LIN {X 0,Y 220.659,Z 422.317,A -85,B 0,C 180,E1 -21894.754,E2 -21894.754} C_VEL
LIN {X 0,Y 216.323,Z 414.128,A -85,B 0,C 180,E1 -21897.374,E2 -21897.374} C_VEL
LIN {X 0,Y 213.162,Z 405.864,A -85,B 0,C 180,E1 -21899.64,E2 -21899.64} C_VEL
LIN {X 0,Y 210.607,Z 397.156,A -85,B 0,C 180,E1 -21901.69,E2 -21901.69} C_VEL
LIN {X 0,Y 207.791,Z 388.841,A -85,B 0,C 180,E1 -21903.524,E2 -21903.524} C_VEL
LIN {X 0,Y 203.956,Z 379.643,A -85,B 0,C 180,E1 -21905.507,E2 -21905.507} C_VEL
LIN {X 0,Y 199.196,Z 370.04,A -85,B 0,C 180,E1 -21907.56,E2 -21907.56} C_VEL
LIN {X 0,Y 195.163,Z 362.8,A -85,B 0,C 180,E1 -21909.133,E2 -21909.133} C_VEL
LIN {X 0,Y 193.052,Z 359.752,A -85,B 0,C 180,E1 -21909.862,E2 -21909.862} C_VEL
LIN {X 0,Y 192.593,Z 357.994,A -85,B 0,C 180,E1 -21910.137,E2 -21910.137} C_VEL
LIN {X 0,Y 192.601,Z 357.995,A -85,B 0,C 180,E1 -21913.892,E2 -21913.892} C_VEL
LIN {X 0,Y 192.582,Z 357.996,A -85,B 0,C 180,E1 -21918.939,E2 -21918.939} C_VEL
LIN {X 0,Y 192.617,Z 357.993,A -85,B 0,C 180,E1 -21923.39,E2 -21923.39} C_VEL
LIN {X 0,Y 192.606,Z 357.992,A -85,B 0,C 180,E1 -21927.06,E2 -21927.06} C_VEL
LIN {X 0,Y 192.663,Z 357.986,A -85,B 0,C 180,E1 -21931.693,E2 -21931.693} C_VEL
LIN {X 0,Y 192.684,Z 357.981,A -85,B 0,C 180,E1 -21936.347,E2 -21936.347} C_VEL
LIN {X 0,Y 192.73,Z 357.974,A -85,B 0,C 180,E1 -21941.46,E2 -21941.46} C_VEL
LIN {X 0,Y 192.771,Z 357.966,A -85,B 0,C 180,E1 -21945.216,E2 -21945.216} C_VEL
LIN {X 0,Y 192.981,Z 357.941,A -85,B 0,C 180,E1 -21949.51,E2 -21949.51} C_VEL
LIN {X 0,Y 193.061,Z 357.934,A -85,B 0,C 180,E1 -21951.628,E2 -21951.628} C_VEL
LIN {X 0,Y 193.263,Z 357.878,A -85,B 0,C 180,E1 -21957.917,E2 -21957.917} C_VEL
LIN {X 0,Y 193.441,Z 357.867,A -85,B 0,C 180,E1 -21960.001,E2 -21960.001} C_VEL
LIN {X 0,Y 192.977,Z 357.947,A -85,B 0,C 180,E1 -21964.178,E2 -21964.178} C_VEL
LIN {X 0,Y 193.062,Z 357.938,A -85,B 0,C 180,E1 -21968.374,E2 -21968.374} C_VEL
LIN {X 0,Y 192.805,Z 357.971,A -85,B 0,C 180,E1 -21972.634,E2 -21972.634} C_VEL
LIN {X 0,Y 192.748,Z 357.978,A -85,B 0,C 180,E1 -21976.961,E2 -21976.961} C_VEL
LIN {X 0,Y 192.612,Z 357.993,A -85,B 0,C 180,E1 -21981.401,E2 -21981.401} C_VEL
LIN {X 0,Y 192.649,Z 357.992,A -85,B 0,C 180,E1 -21984.214,E2 -21984.214} C_VEL
LIN {X 0,Y 192.786,Z 359.362,A -85,B 0,C 180,E1 -21988.965,E2 -21988.965} C_VEL
LIN {X 0,Y 193.005,Z 360.907,A -85,B 0,C 180,E1 -21993.122,E2 -21993.122} C_VEL
LIN {X 0,Y 193.263,Z 362.968,A -85,B 0,C 180,E1 -21998.186,E2 -21998.186} C_VEL
LIN {X 0,Y 193.461,Z 364.155,A -85,B 0,C 180,E1 -22000.838,E2 -22000.838} C_VEL
LIN {X 0,Y 193.547,Z 365.487,A -85,B 0,C 180,E1 -22003.625,E2 -22003.625} C_VEL
LIN {X 0,Y 193.473,Z 367.008,A -85,B 0,C 180,E1 -22006.596,E2 -22006.596} C_VEL
LIN {X 0,Y 193.093,Z 369.197,A -85,B 0,C 180,E1 -22010.252,E2 -22010.252} C_VEL
LIN {X 0,Y 194.095,Z 372.41,A -85,B 0,C 180,E1 -22010.704,E2 -22010.704} C_VEL
LIN {X 0,Y 195.101,Z 374.855,A -85,B 0,C 180,E1 -22011.16,E2 -22011.16} C_VEL
LIN {X 0,Y 198.787,Z 385.581,A -85,B 0,C 180,E1 -22013.057,E2 -22013.057} C_VEL
LIN {X 0,Y 201.301,Z 395.593,A -85,B 0,C 180,E1 -22014.861,E2 -22014.861} C_VEL
LIN {X 0,Y 203.066,Z 406.042,A -85,B 0,C 180,E1 -22016.86,E2 -22016.86} C_VEL
LIN {X 0,Y 203.842,Z 413.828,A -85,B 0,C 180,E1 -22018.453,E2 -22018.453} C_VEL
LIN {X 0,Y 204.14,Z 422.793,A -85,B 0,C 180,E1 -22020.469,E2 -22020.469} C_VEL
LIN {X 0,Y 203.837,Z 430.066,A -85,B 0,C 180,E1 -22022.26,E2 -22022.26} C_VEL
LIN {X 0,Y 200.958,Z 439.204,A -85,B 0,C 180,E1 -22024.633,E2 -22024.633} C_VEL
LIN {X 0,Y 198.837,Z 445.405,A -85,B 0,C 180,E1 -22026.57,E2 -22026.57} C_VEL
LIN {X 0,Y 196.706,Z 451.947,A -85,B 0,C 180,E1 -22029.067,E2 -22029.067} C_VEL
LIN {X 0,Y 195.097,Z 456.448,A -85,B 0,C 180,E1 -22031.083,E2 -22031.083} C_VEL
LIN {X 0,Y 193.055,Z 461.939,A -85,B 0,C 180,E1 -22034.155,E2 -22034.155} C_VEL
LIN {X 0,Y 191.669,Z 466.269,A -85,B 0,C 180,E1 -22037.291,E2 -22037.291} C_VEL
LIN {X 0,Y 191.028,Z 468.641,A -85,B 0,C 180,E1 -22039.4,E2 -22039.4} C_VEL
LIN {X 0,Y 190.544,Z 470.443,A -85,B 0,C 180,E1 -22041.516,E2 -22041.516} C_VEL
LIN {X 0,Y 190.166,Z 472.9,A -85,B 0,C 180,E1 -22045.761,E2 -22045.761} C_VEL
LIN {X 0,Y 190.196,Z 473.608,A -85,B 0,C 180,E1 -22049.408,E2 -22049.408} C_VEL
LIN {X 0,Y 190.148,Z 473.494,A -85,B 0,C 180,E1 -22052.118,E2 -22052.118} C_VEL
LIN {X 0,Y 190.132,Z 472.899,A -85,B 0,C 180,E1 -22054.24,E2 -22054.24} C_VEL
LIN {X 0,Y 190.534,Z 470.478,A -85,B 0,C 180,E1 -22058.432,E2 -22058.432} C_VEL
LIN {X 0,Y 190.229,Z 469.146,A -85,B 0,C 180,E1 -22060.159,E2 -22060.159} C_VEL
LIN {X 0,Y 188.184,Z 466.267,A -85,B 0,C 180,E1 -22062.966,E2 -22062.966} C_VEL
LIN {X 0,Y 186.516,Z 462.684,A -85,B 0,C 180,E1 -22065.759,E2 -22065.759} C_VEL
LIN {X 0,Y 186.811,Z 460.233,A -85,B 0,C 180,E1 -22067.413,E2 -22067.413} C_VEL
LIN {X 0,Y 189.139,Z 454.06,A -85,B 0,C 180,E1 -22070.671,E2 -22070.671} C_VEL
LIN {X 0,Y 191.231,Z 448.498,A -85,B 0,C 180,E1 -22073.048,E2 -22073.048} C_VEL
LIN {X 0,Y 193.396,Z 442.26,A -85,B 0,C 180,E1 -22075.277,E2 -22075.277} C_VEL
LIN {X 0,Y 196.357,Z 433.71,A -85,B 0,C 180,E1 -22077.729,E2 -22077.729} C_VEL
LIN {X 0,Y 197.301,Z 429.862,A -85,B 0,C 180,E1 -22078.743,E2 -22078.743} C_VEL
LIN {X 0,Y 197.649,Z 420.804,A -85,B 0,C 180,E1 -22081.061,E2 -22081.061} C_VEL
LIN {X 0,Y 197.017,Z 409.915,A -85,B 0,C 180,E1 -22083.534,E2 -22083.534} C_VEL
LIN {X 0,Y 195.561,Z 399.633,A -85,B 0,C 180,E1 -22085.667,E2 -22085.667} C_VEL
LIN {X 0,Y 193.558,Z 390.311,A -85,B 0,C 180,E1 -22087.492,E2 -22087.492} C_VEL
LIN {X 0,Y 190.182,Z 379.595,A -85,B 0,C 180,E1 -22089.562,E2 -22089.562} C_VEL
LIN {X 0,Y 187.591,Z 372.854,A -85,B 0,C 180,E1 -22090.884,E2 -22090.884} C_VEL
LIN {X 0,Y 186.322,Z 369.703,A -85,B 0,C 180,E1 -22091.449,E2 -22091.449} C_VEL
LIN {X 0,Y 186.186,Z 368.811,A -85,B 0,C 180,E1 -22091.558,E2 -22091.558} C_VEL
LIN {X 0,Y 186.465,Z 366.674,A -85,B 0,C 180,E1 -22095.735,E2 -22095.735} C_VEL
LIN {X 0,Y 186.364,Z 364.657,A -85,B 0,C 180,E1 -22100.125,E2 -22100.125} C_VEL
LIN {X 0,Y 186.017,Z 362.453,A -85,B 0,C 180,E1 -22105.477,E2 -22105.477} C_VEL
LIN {X 0,Y 185.791,Z 360.632,A -85,B 0,C 180,E1 -22110.543,E2 -22110.543} C_VEL
LIN {X 0,Y 185.626,Z 359.083,A -85,B 0,C 180,E1 -22115.387,E2 -22115.387} C_VEL
LIN {X 0,Y 185.673,Z 358.859,A -85,B 0,C 180,E1 -22121.134,E2 -22121.134} C_VEL
LIN {X 0,Y 185.729,Z 358.85,A -85,B 0,C 180,E1 -22126.876,E2 -22126.876} C_VEL
LIN {X 0,Y 186.009,Z 358.817,A -85,B 0,C 180,E1 -22131.306,E2 -22131.306} C_VEL
LIN {X 0,Y 186.208,Z 358.787,A -85,B 0,C 180,E1 -22137.836,E2 -22137.836} C_VEL
LIN {X 0,Y 186.405,Z 358.742,A -85,B 0,C 180,E1 -22139.999,E2 -22139.999} C_VEL
LIN {X 0,Y 185.923,Z 358.812,A -85,B 0,C 180,E1 -22144.335,E2 -22144.335} C_VEL
LIN {X 0,Y 186.008,Z 358.81,A -85,B 0,C 180,E1 -22148.691,E2 -22148.691} C_VEL
LIN {X 0,Y 185.764,Z 358.843,A -85,B 0,C 180,E1 -22153.119,E2 -22153.119} C_VEL
LIN {X 0,Y 185.672,Z 358.851,A -85,B 0,C 180,E1 -22158.864,E2 -22158.864} C_VEL
LIN {X 0,Y 185.575,Z 358.861,A -85,B 0,C 180,E1 -22164.645,E2 -22164.645} C_VEL
LIN {X 0,Y 185.577,Z 358.868,A -85,B 0,C 180,E1 -22169.492,E2 -22169.492} C_VEL
LIN {X 0,Y 185.519,Z 358.877,A -85,B 0,C 180,E1 -22174.626,E2 -22174.626} C_VEL
LIN {X 0,Y 185.566,Z 358.87,A -85,B 0,C 180,E1 -22177.313,E2 -22177.313} C_VEL
LIN {X 0,Y 185.559,Z 358.87,A -85,B 0,C 180,E1 -22180.757,E2 -22180.757} C_VEL
LIN {X 0,Y 185.561,Z 358.872,A -85,B 0,C 180,E1 -22186.021,E2 -22186.021} C_VEL
LIN {X 0,Y 185.518,Z 358.882,A -85,B 0,C 180,E1 -22188.115,E2 -22188.115} C_VEL
LIN {X 0,Y 186.432,Z 361.575,A -85,B 0,C 180,E1 -22188.552,E2 -22188.552} C_VEL
LIN {X 0,Y 188.38,Z 364.16,A -85,B 0,C 180,E1 -22189.253,E2 -22189.253} C_VEL
LIN {X 0,Y 193,Z 372.328,A -85,B 0,C 180,E1 -22191.213,E2 -22191.213} C_VEL
LIN {X 0,Y 198.325,Z 383.032,A -85,B 0,C 180,E1 -22193.722,E2 -22193.722} C_VEL
LIN {X 0,Y 202.66,Z 394.236,A -85,B 0,C 180,E1 -22196.332,E2 -22196.332} C_VEL
LIN {X 0,Y 205.561,Z 404.141,A -85,B 0,C 180,E1 -22198.728,E2 -22198.728} C_VEL
LIN {X 0,Y 208.189,Z 412.696,A -85,B 0,C 180,E1 -22201.047,E2 -22201.047} C_VEL
LIN {X 0,Y 210.839,Z 419.24,A -85,B 0,C 180,E1 -22203.08,E2 -22203.08} C_VEL
LIN {X 0,Y 215.488,Z 427.187,A -85,B 0,C 180,E1 -22205.948,E2 -22205.948} C_VEL
LIN {X 0,Y 221.572,Z 434.829,A -85,B 0,C 180,E1 -22209.137,E2 -22209.137} C_VEL
LIN {X 0,Y 228.686,Z 441.416,A -85,B 0,C 180,E1 -22212.303,E2 -22212.303} C_VEL
LIN {X 0,Y 236.191,Z 446.779,A -85,B 0,C 180,E1 -22215.245,E2 -22215.245} C_VEL
LIN {X 0,Y 244.931,Z 451.783,A -85,B 0,C 180,E1 -22218.413,E2 -22218.413} C_VEL
LIN {X 0,Y 252.724,Z 455.469,A -85,B 0,C 180,E1 -22221.202,E2 -22221.202} C_VEL
LIN {X 0,Y 259.303,Z 458.169,A -85,B 0,C 180,E1 -22223.776,E2 -22223.776} C_VEL
LIN {X 0,Y 262.787,Z 459.443,A -85,B 0,C 180,E1 -22225.398,E2 -22225.398} C_VEL
LIN {X 0,Y 265.271,Z 460.379,A -85,B 0,C 180,E1 -22226.963,E2 -22226.963} C_VEL
LIN {X 0,Y 267.516,Z 460.902,A -85,B 0,C 180,E1 -22228.495,E2 -22228.495} C_VEL
LIN {X 0,Y 268.92,Z 461.053,A -85,B 0,C 180,E1 -22230,E2 -22230} C_VEL
LIN {X 0,Y 267.179,Z 460.84,A -85,B 0,C 180,E1 -22231.715,E2 -22231.715} C_VEL
LIN {X 0,Y 265.224,Z 460.38,A -85,B 0,C 180,E1 -22233.038,E2 -22233.038} C_VEL
LIN {X 0,Y 262.759,Z 459.444,A -85,B 0,C 180,E1 -22234.602,E2 -22234.602} C_VEL
LIN {X 0,Y 259.293,Z 458.17,A -85,B 0,C 180,E1 -22236.224,E2 -22236.224} C_VEL
LIN {X 0,Y 255.099,Z 456.489,A -85,B 0,C 180,E1 -22237.918,E2 -22237.918} C_VEL
LIN {X 0,Y 247.647,Z 453.148,A -85,B 0,C 180,E1 -22240.633,E2 -22240.633} C_VEL
LIN {X 0,Y 238.803,Z 448.431,A -85,B 0,C 180,E1 -22243.79,E2 -22243.79} C_VEL
LIN {X 0,Y 231.132,Z 443.335,A -85,B 0,C 180,E1 -22246.705,E2 -22246.705} C_VEL
LIN {X 0,Y 223.99,Z 437.284,A -85,B 0,C 180,E1 -22249.733,E2 -22249.733} C_VEL
LIN {X 0,Y 217.685,Z 430.326,A -85,B 0,C 180,E1 -22252.794,E2 -22252.794} C_VEL
LIN {X 0,Y 212.841,Z 422.953,A -85,B 0,C 180,E1 -22255.616,E2 -22255.616} C_VEL
LIN {X 0,Y 209.307,Z 415.708,A -85,B 0,C 180,E1 -22258.04,E2 -22258.04} C_VEL
LIN {X 0,Y 206.487,Z 407.564,A -85,B 0,C 180,E1 -22260.382,E2 -22260.382} C_VEL
LIN {X 0,Y 203.788,Z 397.831,A -85,B 0,C 180,E1 -22262.797,E2 -22262.797} C_VEL
LIN {X 0,Y 200.962,Z 389.663,A -85,B 0,C 180,E1 -22264.731,E2 -22264.731} C_VEL
LIN {X 0,Y 197.354,Z 380.929,A -85,B 0,C 180,E1 -22266.752,E2 -22266.752} C_VEL
LIN {X 0,Y 192.359,Z 371.004,A -85,B 0,C 180,E1 -22269.071,E2 -22269.071} C_VEL
LIN {X 0,Y 188.188,Z 363.769,A -85,B 0,C 180,E1 -22270.828,E2 -22270.828} C_VEL
LIN {X 0,Y 186.069,Z 360.806,A -85,B 0,C 180,E1 -22271.623,E2 -22271.623} C_VEL
LIN {X 0,Y 185.527,Z 358.875,A -85,B 0,C 180,E1 -22271.963,E2 -22271.963} C_VEL
LIN {X 0,Y 185.555,Z 358.87,A -85,B 0,C 180,E1 -22277.02,E2 -22277.02} C_VEL
LIN {X 0,Y 185.539,Z 358.873,A -85,B 0,C 180,E1 -22279.915,E2 -22279.915} C_VEL
LIN {X 0,Y 185.557,Z 358.871,A -85,B 0,C 180,E1 -22282.701,E2 -22282.701} C_VEL
LIN {X 0,Y 185.544,Z 358.873,A -85,B 0,C 180,E1 -22287.976,E2 -22287.976} C_VEL
LIN {X 0,Y 185.58,Z 358.868,A -85,B 0,C 180,E1 -22290.577,E2 -22290.577} C_VEL
LIN {X 0,Y 185.578,Z 358.861,A -85,B 0,C 180,E1 -22295.383,E2 -22295.383} C_VEL
LIN {X 0,Y 185.672,Z 358.851,A -85,B 0,C 180,E1 -22301.136,E2 -22301.136} C_VEL
LIN {X 0,Y 185.764,Z 358.843,A -85,B 0,C 180,E1 -22306.881,E2 -22306.881} C_VEL
LIN {X 0,Y 186.008,Z 358.81,A -85,B 0,C 180,E1 -22311.309,E2 -22311.309} C_VEL
LIN {X 0,Y 186.207,Z 358.756,A -85,B 0,C 180,E1 -22317.838,E2 -22317.838} C_VEL
LIN {X 0,Y 186.405,Z 358.742,A -85,B 0,C 180,E1 -22320.001,E2 -22320.001} C_VEL
LIN {X 0,Y 185.925,Z 358.826,A -85,B 0,C 180,E1 -22324.337,E2 -22324.337} C_VEL
LIN {X 0,Y 186.009,Z 358.816,A -85,B 0,C 180,E1 -22328.694,E2 -22328.694} C_VEL
LIN {X 0,Y 185.729,Z 358.852,A -85,B 0,C 180,E1 -22333.124,E2 -22333.124} C_VEL
LIN {X 0,Y 185.673,Z 358.858,A -85,B 0,C 180,E1 -22338.866,E2 -22338.866} C_VEL
LIN {X 0,Y 185.626,Z 359.073,A -85,B 0,C 180,E1 -22344.613,E2 -22344.613} C_VEL
LIN {X 0,Y 185.786,Z 360.66,A -85,B 0,C 180,E1 -22349.535,E2 -22349.535} C_VEL
LIN {X 0,Y 186.017,Z 362.452,A -85,B 0,C 180,E1 -22354.523,E2 -22354.523} C_VEL
LIN {X 0,Y 186.366,Z 364.652,A -85,B 0,C 180,E1 -22359.874,E2 -22359.874} C_VEL
LIN {X 0,Y 186.463,Z 366.673,A -85,B 0,C 180,E1 -22364.264,E2 -22364.264} C_VEL
LIN {X 0,Y 186.189,Z 368.886,A -85,B 0,C 180,E1 -22368.457,E2 -22368.457} C_VEL
LIN {X 0,Y 187.079,Z 371.908,A -85,B 0,C 180,E1 -22368.903,E2 -22368.903} C_VEL
LIN {X 0,Y 188.338,Z 374.524,A -85,B 0,C 180,E1 -22369.474,E2 -22369.474} C_VEL
LIN {X 0,Y 192.135,Z 385.349,A -85,B 0,C 180,E1 -22371.55,E2 -22371.55} C_VEL
LIN {X 0,Y 194.4,Z 393.639,A -85,B 0,C 180,E1 -22373.143,E2 -22373.143} C_VEL
LIN {X 0,Y 196.393,Z 404.84,A -85,B 0,C 180,E1 -22375.394,E2 -22375.394} C_VEL
LIN {X 0,Y 197.326,Z 413.913,A -85,B 0,C 180,E1 -22377.35,E2 -22377.35} C_VEL
LIN {X 0,Y 197.597,Z 423.15,A -85,B 0,C 180,E1 -22379.535,E2 -22379.535} C_VEL
LIN {X 0,Y 197.309,Z 429.862,A -85,B 0,C 180,E1 -22381.259,E2 -22381.259} C_VEL
LIN {X 0,Y 196.387,Z 433.711,A -85,B 0,C 180,E1 -22382.275,E2 -22382.275} C_VEL
LIN {X 0,Y 193.415,Z 442.261,A -85,B 0,C 180,E1 -22384.726,E2 -22384.726} C_VEL
LIN {X 0,Y 190.835,Z 449.823,A -85,B 0,C 180,E1 -22387.459,E2 -22387.459} C_VEL
LIN {X 0,Y 188.349,Z 456.251,A -85,B 0,C 180,E1 -22390.378,E2 -22390.378} C_VEL
LIN {X 0,Y 186.208,Z 461.743,A -85,B 0,C 180,E1 -22393.557,E2 -22393.557} C_VEL
LIN {X 0,Y 184.726,Z 466.073,A -85,B 0,C 180,E1 -22396.805,E2 -22396.805} C_VEL
LIN {X 0,Y 184.036,Z 468.444,A -85,B 0,C 180,E1 -22398.992,E2 -22398.992} C_VEL
LIN {X 0,Y 183.514,Z 470.247,A -85,B 0,C 180,E1 -22401.188,E2 -22401.188} C_VEL
LIN {X 0,Y 183.08,Z 472.704,A -85,B 0,C 180,E1 -22405.597,E2 -22405.597} C_VEL
LIN {X 0,Y 183.052,Z 473.298,A -85,B 0,C 180,E1 -22407.8,E2 -22407.8} C_VEL
LIN {X 0,Y 183.154,Z 473.457,A -85,B 0,C 180,E1 -22410,E2 -22410} C_VEL
LIN {X 0,Y 183.02,Z 473.024,A -85,B 0,C 180,E1 -22413.216,E2 -22413.216} C_VEL
LIN {X 0,Y 183.215,Z 471.64,A -85,B 0,C 180,E1 -22416.608,E2 -22416.608} C_VEL
LIN {X 0,Y 183.513,Z 470.247,A -85,B 0,C 180,E1 -22418.812,E2 -22418.812} C_VEL
LIN {X 0,Y 184.34,Z 467.291,A -85,B 0,C 180,E1 -22422.104,E2 -22422.104} C_VEL
LIN {X 0,Y 185.597,Z 463.296,A -85,B 0,C 180,E1 -22425.371,E2 -22425.371} C_VEL
LIN {X 0,Y 186.811,Z 460.233,A -85,B 0,C 180,E1 -22427.413,E2 -22427.413} C_VEL
LIN {X 0,Y 187.234,Z 457.581,A -85,B 0,C 180,E1 -22429.026,E2 -22429.026} C_VEL
LIN {X 0,Y 186.33,Z 452.716,A -85,B 0,C 180,E1 -22431.665,E2 -22431.665} C_VEL
LIN {X 0,Y 185.641,Z 447.322,A -85,B 0,C 180,E1 -22434.225,E2 -22434.225} C_VEL
LIN {X 0,Y 186.393,Z 443.699,A -85,B 0,C 180,E1 -22435.666,E2 -22435.666} C_VEL
LIN {X 0,Y 189.413,Z 435.432,A -85,B 0,C 180,E1 -22438.234,E2 -22438.234} C_VEL
LIN {X 0,Y 190.569,Z 431.589,A -85,B 0,C 180,E1 -22439.251,E2 -22439.251} C_VEL
LIN {X 0,Y 191.068,Z 425.28,A -85,B 0,C 180,E1 -22440.995,E2 -22440.995} C_VEL
LIN {X 0,Y 191.074,Z 417.952,A -85,B 0,C 180,E1 -22442.878,E2 -22442.878} C_VEL
LIN {X 0,Y 190.367,Z 407.971,A -85,B 0,C 180,E1 -22445.208,E2 -22445.208} C_VEL
LIN {X 0,Y 188.967,Z 398.666,A -85,B 0,C 180,E1 -22447.237,E2 -22447.237} C_VEL
LIN {X 0,Y 186.873,Z 389.688,A -85,B 0,C 180,E1 -22449.134,E2 -22449.134} C_VEL
LIN {X 0,Y 183.639,Z 379.656,A -85,B 0,C 180,E1 -22451.239,E2 -22451.239} C_VEL
LIN {X 0,Y 180.903,Z 372.89,A -85,B 0,C 180,E1 -22452.716,E2 -22452.716} C_VEL
LIN {X 0,Y 179.565,Z 369.943,A -85,B 0,C 180,E1 -22453.347,E2 -22453.347} C_VEL
LIN {X 0,Y 179.31,Z 368.567,A -85,B 0,C 180,E1 -22453.557,E2 -22453.557} C_VEL
LIN {X 0,Y 179.373,Z 366.418,A -85,B 0,C 180,E1 -22458.234,E2 -22458.234} C_VEL
LIN {X 0,Y 179.196,Z 364.965,A -85,B 0,C 180,E1 -22461.664,E2 -22461.664} C_VEL
LIN {X 0,Y 178.921,Z 363.024,A -85,B 0,C 180,E1 -22466.637,E2 -22466.637} C_VEL
LIN {X 0,Y 178.677,Z 361.274,A -85,B 0,C 180,E1 -22471.834,E2 -22471.834} C_VEL
LIN {X 0,Y 178.51,Z 359.807,A -85,B 0,C 180,E1 -22476.814,E2 -22476.814} C_VEL
LIN {X 0,Y 178.647,Z 359.734,A -85,B 0,C 180,E1 -22481.655,E2 -22481.655} C_VEL
LIN {X 0,Y 178.655,Z 359.731,A -85,B 0,C 180,E1 -22486.346,E2 -22486.346} C_VEL
LIN {X 0,Y 178.96,Z 359.694,A -85,B 0,C 180,E1 -22490.961,E2 -22490.961} C_VEL
LIN {X 0,Y 179.154,Z 359.665,A -85,B 0,C 180,E1 -22497.751,E2 -22497.751} C_VEL
LIN {X 0,Y 179.368,Z 359.617,A -85,B 0,C 180,E1 -22499.999,E2 -22499.999} C_VEL
LIN {X 0,Y 178.872,Z 359.691,A -85,B 0,C 180,E1 -22504.506,E2 -22504.506} C_VEL
LIN {X 0,Y 178.937,Z 359.688,A -85,B 0,C 180,E1 -22509.038,E2 -22509.038} C_VEL
LIN {X 0,Y 178.681,Z 359.724,A -85,B 0,C 180,E1 -22513.649,E2 -22513.649} C_VEL
LIN {X 0,Y 178.62,Z 359.728,A -85,B 0,C 180,E1 -22519.213,E2 -22519.213} C_VEL
LIN {X 0,Y 178.518,Z 359.74,A -85,B 0,C 180,E1 -22525.113,E2 -22525.113} C_VEL
LIN {X 0,Y 178.521,Z 359.748,A -85,B 0,C 180,E1 -22529.993,E2 -22529.993} C_VEL
LIN {X 0,Y 178.483,Z 359.752,A -85,B 0,C 180,E1 -22534.219,E2 -22534.219} C_VEL
LIN {X 0,Y 178.47,Z 359.754,A -85,B 0,C 180,E1 -22539.053,E2 -22539.053} C_VEL
LIN {X 0,Y 178.497,Z 359.751,A -85,B 0,C 180,E1 -22542.015,E2 -22542.015} C_VEL
LIN {X 0,Y 178.538,Z 359.816,A -85,B 0,C 180,E1 -22546.123,E2 -22546.123} C_VEL
LIN {X 0,Y 179.475,Z 362.544,A -85,B 0,C 180,E1 -22546.612,E2 -22546.612} C_VEL
LIN {X 0,Y 181.331,Z 364.906,A -85,B 0,C 180,E1 -22547.347,E2 -22547.347} C_VEL
LIN {X 0,Y 183.395,Z 368.391,A -85,B 0,C 180,E1 -22548.309,E2 -22548.309} C_VEL
LIN {X 0,Y 187.7,Z 376.009,A -85,B 0,C 180,E1 -22550.302,E2 -22550.302} C_VEL
LIN {X 0,Y 192.54,Z 386.219,A -85,B 0,C 180,E1 -22552.904,E2 -22552.904} C_VEL
LIN {X 0,Y 196.289,Z 396.271,A -85,B 0,C 180,E1 -22555.435,E2 -22555.435} C_VEL
LIN {X 0,Y 198.802,Z 404.826,A -85,B 0,C 180,E1 -22557.644,E2 -22557.644} C_VEL
LIN {X 0,Y 201.278,Z 414.124,A -85,B 0,C 180,E1 -22560.266,E2 -22560.266} C_VEL
LIN {X 0,Y 204.171,Z 421.72,A -85,B 0,C 180,E1 -22562.775,E2 -22562.775} C_VEL
LIN {X 0,Y 208.311,Z 429.129,A -85,B 0,C 180,E1 -22565.631,E2 -22565.631} C_VEL
LIN {X 0,Y 213.87,Z 436.283,A -85,B 0,C 180,E1 -22568.81,E2 -22568.81} C_VEL
LIN {X 0,Y 221.275,Z 443.146,A -85,B 0,C 180,E1 -22572.331,E2 -22572.331} C_VEL
LIN {X 0,Y 229.894,Z 449.032,A -85,B 0,C 180,E1 -22575.844,E2 -22575.844} C_VEL
LIN {X 0,Y 236.751,Z 452.702,A -85,B 0,C 180,E1 -22578.405,E2 -22578.405} C_VEL
LIN {X 0,Y 242.334,Z 455.19,A -85,B 0,C 180,E1 -22580.41,E2 -22580.41} C_VEL
LIN {X 0,Y 248.081,Z 457.466,A -85,B 0,C 180,E1 -22582.53,E2 -22582.53} C_VEL
LIN {X 0,Y 254.811,Z 459.662,A -85,B 0,C 180,E1 -22585.254,E2 -22585.254} C_VEL
LIN {X 0,Y 257.632,Z 460.592,A -85,B 0,C 180,E1 -22586.872,E2 -22586.872} C_VEL
LIN {X 0,Y 260.119,Z 461.125,A -85,B 0,C 180,E1 -22588.514,E2 -22588.514} C_VEL
LIN {X 0,Y 261.658,Z 461.25,A -85,B 0,C 180,E1 -22590,E2 -22590} C_VEL
LIN {X 0,Y 259.965,Z 461.109,A -85,B 0,C 180,E1 -22591.549,E2 -22591.549} C_VEL
LIN {X 0,Y 257.576,Z 460.592,A -85,B 0,C 180,E1 -22593.128,E2 -22593.128} C_VEL
LIN {X 0,Y 254.007,Z 459.433,A -85,B 0,C 180,E1 -22595.094,E2 -22595.094} C_VEL
LIN {X 0,Y 248.095,Z 457.438,A -85,B 0,C 180,E1 -22597.494,E2 -22597.494} C_VEL
LIN {X 0,Y 240.998,Z 454.618,A -85,B 0,C 180,E1 -22600.077,E2 -22600.077} C_VEL
LIN {X 0,Y 231.366,Z 449.896,A -85,B 0,C 180,E1 -22603.587,E2 -22603.587} C_VEL
LIN {X 0,Y 223.415,Z 444.784,A -85,B 0,C 180,E1 -22606.758,E2 -22606.758} C_VEL
LIN {X 0,Y 216.641,Z 439.112,A -85,B 0,C 180,E1 -22609.82,E2 -22609.82} C_VEL
LIN {X 0,Y 210.259,Z 431.926,A -85,B 0,C 180,E1 -22613.196,E2 -22613.196} C_VEL
LIN {X 0,Y 205.27,Z 423.882,A -85,B 0,C 180,E1 -22616.429,E2 -22616.429} C_VEL
LIN {X 0,Y 201.894,Z 415.933,A -85,B 0,C 180,E1 -22619.166,E2 -22619.166} C_VEL
LIN {X 0,Y 199.303,Z 407.067,A -85,B 0,C 180,E1 -22621.761,E2 -22621.761} C_VEL
LIN {X 0,Y 197.169,Z 398.915,A -85,B 0,C 180,E1 -22623.878,E2 -22623.878} C_VEL
LIN {X 0,Y 193.866,Z 389.659,A -85,B 0,C 180,E1 -22626.236,E2 -22626.236} C_VEL
LIN {X 0,Y 190.688,Z 382.257,A -85,B 0,C 180,E1 -22628.117,E2 -22628.117} C_VEL
LIN {X 0,Y 185.633,Z 372.173,A -85,B 0,C 180,E1 -22630.681,E2 -22630.681} C_VEL
LIN {X 0,Y 182.496,Z 367.228,A -85,B 0,C 180,E1 -22632.071,E2 -22632.071} C_VEL
LIN {X 0,Y 180.834,Z 364.144,A -85,B 0,C 180,E1 -22632.864,E2 -22632.864} C_VEL
LIN {X 0,Y 179.125,Z 361.888,A -85,B 0,C 180,E1 -22633.564,E2 -22633.564} C_VEL
LIN {X 0,Y 178.518,Z 359.749,A -85,B 0,C 180,E1 -22633.972,E2 -22633.972} C_VEL
LIN {X 0,Y 178.5,Z 359.751,A -85,B 0,C 180,E1 -22638.424,E2 -22638.424} C_VEL
LIN {X 0,Y 178.457,Z 359.755,A -85,B 0,C 180,E1 -22643.793,E2 -22643.793} C_VEL
LIN {X 0,Y 178.489,Z 359.749,A -85,B 0,C 180,E1 -22646.549,E2 -22646.549} C_VEL
LIN {X 0,Y 178.521,Z 359.748,A -85,B 0,C 180,E1 -22650.007,E2 -22650.007} C_VEL
LIN {X 0,Y 178.518,Z 359.74,A -85,B 0,C 180,E1 -22654.887,E2 -22654.887} C_VEL
LIN {X 0,Y 178.62,Z 359.728,A -85,B 0,C 180,E1 -22660.787,E2 -22660.787} C_VEL
LIN {X 0,Y 178.681,Z 359.724,A -85,B 0,C 180,E1 -22666.351,E2 -22666.351} C_VEL
LIN {X 0,Y 178.937,Z 359.688,A -85,B 0,C 180,E1 -22670.962,E2 -22670.962} C_VEL
LIN {X 0,Y 179.153,Z 359.634,A -85,B 0,C 180,E1 -22677.753,E2 -22677.753} C_VEL
LIN {X 0,Y 179.368,Z 359.617,A -85,B 0,C 180,E1 -22680.001,E2 -22680.001} C_VEL
LIN {X 0,Y 178.873,Z 359.704,A -85,B 0,C 180,E1 -22684.508,E2 -22684.508} C_VEL
LIN {X 0,Y 178.96,Z 359.694,A -85,B 0,C 180,E1 -22689.039,E2 -22689.039} C_VEL
LIN {X 0,Y 178.655,Z 359.733,A -85,B 0,C 180,E1 -22693.654,E2 -22693.654} C_VEL
LIN {X 0,Y 178.621,Z 359.736,A -85,B 0,C 180,E1 -22699.214,E2 -22699.214} C_VEL
LIN {X 0,Y 178.511,Z 359.807,A -85,B 0,C 180,E1 -22703.186,E2 -22703.186} C_VEL
LIN {X 0,Y 178.687,Z 361.271,A -85,B 0,C 180,E1 -22708.164,E2 -22708.164} C_VEL
LIN {X 0,Y 178.918,Z 363.016,A -85,B 0,C 180,E1 -22713.363,E2 -22713.363} C_VEL
LIN {X 0,Y 179.229,Z 365.174,A -85,B 0,C 180,E1 -22718.86,E2 -22718.86} C_VEL
LIN {X 0,Y 179.385,Z 366.469,A -85,B 0,C 180,E1 -22721.894,E2 -22721.894} C_VEL
LIN {X 0,Y 179.301,Z 368.595,A -85,B 0,C 180,E1 -22726.445,E2 -22726.445} C_VEL
LIN {X 0,Y 180.276,Z 371.801,A -85,B 0,C 180,E1 -22727.001,E2 -22727.001} C_VEL
LIN {X 0,Y 181.562,Z 374.368,A -85,B 0,C 180,E1 -22727.63,E2 -22727.63} C_VEL
LIN {X 0,Y 184.468,Z 381.628,A -85,B 0,C 180,E1 -22729.186,E2 -22729.186} C_VEL
LIN {X 0,Y 187.999,Z 393.775,A -85,B 0,C 180,E1 -22731.727,E2 -22731.727} C_VEL
LIN {X 0,Y 189.898,Z 404.623,A -85,B 0,C 180,E1 -22734.031,E2 -22734.031} C_VEL
LIN {X 0,Y 190.858,Z 413.994,A -85,B 0,C 180,E1 -22736.165,E2 -22736.165} C_VEL
LIN {X 0,Y 191.157,Z 421.739,A -85,B 0,C 180,E1 -22738.067,E2 -22738.067} C_VEL
LIN {X 0,Y 190.842,Z 429.657,A -85,B 0,C 180,E1 -22740.188,E2 -22740.188} C_VEL
LIN {X 0,Y 190.105,Z 433.514,A -85,B 0,C 180,E1 -22741.276,E2 -22741.276} C_VEL
LIN {X 0,Y 186.979,Z 442.064,A -85,B 0,C 180,E1 -22743.791,E2 -22743.791} C_VEL
LIN {X 0,Y 183.967,Z 450.371,A -85,B 0,C 180,E1 -22746.933,E2 -22746.933} C_VEL
LIN {X 0,Y 181.625,Z 456.054,A -85,B 0,C 180,E1 -22749.619,E2 -22749.619} C_VEL
LIN {X 0,Y 179.388,Z 461.546,A -85,B 0,C 180,E1 -22752.913,E2 -22752.913} C_VEL
LIN {X 0,Y 177.781,Z 465.876,A -85,B 0,C 180,E1 -22756.279,E2 -22756.279} C_VEL
LIN {X 0,Y 177.032,Z 468.247,A -85,B 0,C 180,E1 -22758.551,E2 -22758.551} C_VEL
LIN {X 0,Y 176.476,Z 470.051,A -85,B 0,C 180,E1 -22760.834,E2 -22760.834} C_VEL
LIN {X 0,Y 176.01,Z 472.509,A -85,B 0,C 180,E1 -22765.42,E2 -22765.42} C_VEL
LIN {X 0,Y 175.972,Z 473.102,A -85,B 0,C 180,E1 -22767.711,E2 -22767.711} C_VEL
LIN {X 0,Y 176.062,Z 473.261,A -85,B 0,C 180,E1 -22770,E2 -22770} C_VEL
LIN {X 0,Y 175.95,Z 472.909,A -85,B 0,C 180,E1 -22773.037,E2 -22773.037} C_VEL
LIN {X 0,Y 176.143,Z 471.444,A -85,B 0,C 180,E1 -22776.875,E2 -22776.875} C_VEL
LIN {X 0,Y 176.476,Z 470.051,A -85,B 0,C 180,E1 -22779.166,E2 -22779.166} C_VEL
LIN {X 0,Y 177.389,Z 467.095,A -85,B 0,C 180,E1 -22782.586,E2 -22782.586} C_VEL
LIN {X 0,Y 178.728,Z 463.1,A -85,B 0,C 180,E1 -22785.977,E2 -22785.977} C_VEL
LIN {X 0,Y 180.865,Z 457.971,A -85,B 0,C 180,E1 -22789.286,E2 -22789.286} C_VEL
LIN {X 0,Y 182.998,Z 452.709,A -85,B 0,C 180,E1 -22791.99,E2 -22791.99} C_VEL
LIN {X 0,Y 185.355,Z 446.389,A -85,B 0,C 180,E1 -22794.65,E2 -22794.65} C_VEL
LIN {X 0,Y 186.393,Z 443.699,A -85,B 0,C 180,E1 -22795.666,E2 -22795.666} C_VEL
LIN {X 0,Y 187.174,Z 439.956,A -85,B 0,C 180,E1 -22797.054,E2 -22797.054} C_VEL
LIN {X 0,Y 186.969,Z 436.113,A -85,B 0,C 180,E1 -22798.447,E2 -22798.447} C_VEL
LIN {X 0,Y 185.327,Z 428.2,A -85,B 0,C 180,E1 -22801.196,E2 -22801.196} C_VEL
LIN {X 0,Y 184.689,Z 422.37,A -85,B 0,C 180,E1 -22802.953,E2 -22802.953} C_VEL
LIN {X 0,Y 184.366,Z 412.255,A -85,B 0,C 180,E1 -22805.571,E2 -22805.571} C_VEL
LIN {X 0,Y 182.883,Z 400.26,A -85,B 0,C 180,E1 -22808.387,E2 -22808.387} C_VEL
LIN {X 0,Y 180.617,Z 390.342,A -85,B 0,C 180,E1 -22810.643,E2 -22810.643} C_VEL
LIN {X 0,Y 177.709,Z 381.192,A -85,B 0,C 180,E1 -22812.744,E2 -22812.744} C_VEL
LIN {X 0,Y 174.712,Z 373.764,A -85,B 0,C 180,E1 -22814.493,E2 -22814.493} C_VEL
LIN {X 0,Y 172.804,Z 370.323,A -85,B 0,C 180,E1 -22815.452,E2 -22815.452} C_VEL
LIN {X 0,Y 172.312,Z 368.302,A -85,B 0,C 180,E1 -22815.853,E2 -22815.853} C_VEL
LIN {X 0,Y 172.196,Z 366.237,A -85,B 0,C 180,E1 -22820.847,E2 -22820.847} C_VEL
LIN {X 0,Y 171.977,Z 364.623,A -85,B 0,C 180,E1 -22825.1,E2 -22825.1} C_VEL
LIN {X 0,Y 171.688,Z 362.73,A -85,B 0,C 180,E1 -22830.578,E2 -22830.578} C_VEL
LIN {X 0,Y 171.519,Z 361.196,A -85,B 0,C 180,E1 -22835.81,E2 -22835.81} C_VEL
LIN {X 0,Y 171.455,Z 360.631,A -85,B 0,C 180,E1 -22838.35,E2 -22838.35} C_VEL
LIN {X 0,Y 171.577,Z 360.615,A -85,B 0,C 180,E1 -22840.87,E2 -22840.87} C_VEL
LIN {X 0,Y 171.572,Z 360.614,A -85,B 0,C 180,E1 -22845.771,E2 -22845.771} C_VEL
LIN {X 0,Y 171.889,Z 360.574,A -85,B 0,C 180,E1 -22850.586,E2 -22850.586} C_VEL
LIN {X 0,Y 171.822,Z 360.581,A -85,B 0,C 180,E1 -22855.306,E2 -22855.306} C_VEL
LIN {X 0,Y 172.331,Z 360.491,A -85,B 0,C 180,E1 -22859.999,E2 -22859.999} C_VEL
LIN {X 0,Y 171.821,Z 360.57,A -85,B 0,C 180,E1 -22864.691,E2 -22864.691} C_VEL
LIN {X 0,Y 171.873,Z 360.567,A -85,B 0,C 180,E1 -22869.412,E2 -22869.412} C_VEL
LIN {X 0,Y 171.593,Z 360.603,A -85,B 0,C 180,E1 -22874.224,E2 -22874.224} C_VEL
LIN {X 0,Y 171.539,Z 360.608,A -85,B 0,C 180,E1 -22879.557,E2 -22879.557} C_VEL
LIN {X 0,Y 171.457,Z 360.621,A -85,B 0,C 180,E1 -22885.608,E2 -22885.608} C_VEL
LIN {X 0,Y 171.44,Z 360.629,A -85,B 0,C 180,E1 -22890.586,E2 -22890.586} C_VEL
LIN {X 0,Y 171.402,Z 360.634,A -85,B 0,C 180,E1 -22895.031,E2 -22895.031} C_VEL
LIN {X 0,Y 171.425,Z 360.632,A -85,B 0,C 180,E1 -22898.835,E2 -22898.835} C_VEL
LIN {X 0,Y 171.423,Z 360.633,A -85,B 0,C 180,E1 -22903.817,E2 -22903.817} C_VEL
LIN {X 0,Y 172.31,Z 363.262,A -85,B 0,C 180,E1 -22904.35,E2 -22904.35} C_VEL
LIN {X 0,Y 174.485,Z 365.931,A -85,B 0,C 180,E1 -22905.321,E2 -22905.321} C_VEL
LIN {X 0,Y 176.415,Z 369.271,A -85,B 0,C 180,E1 -22906.326,E2 -22906.326} C_VEL
LIN {X 0,Y 181.182,Z 377.441,A -85,B 0,C 180,E1 -22908.744,E2 -22908.744} C_VEL
LIN {X 0,Y 185.866,Z 387.378,A -85,B 0,C 180,E1 -22911.495,E2 -22911.495} C_VEL
LIN {X 0,Y 189.215,Z 396.204,A -85,B 0,C 180,E1 -22913.885,E2 -22913.885} C_VEL
LIN {X 0,Y 191.851,Z 404.715,A -85,B 0,C 180,E1 -22916.24,E2 -22916.24} C_VEL
LIN {X 0,Y 194.215,Z 414.654,A -85,B 0,C 180,E1 -22919.153,E2 -22919.153} C_VEL
LIN {X 0,Y 197.045,Z 423.08,A -85,B 0,C 180,E1 -22922.055,E2 -22922.055} C_VEL
LIN {X 0,Y 200.147,Z 429.245,A -85,B 0,C 180,E1 -22924.524,E2 -22924.524} C_VEL
LIN {X 0,Y 205.215,Z 436.533,A -85,B 0,C 180,E1 -22927.87,E2 -22927.87} C_VEL
LIN {X 0,Y 209.945,Z 441.457,A -85,B 0,C 180,E1 -22930.443,E2 -22930.443} C_VEL
LIN {X 0,Y 216.399,Z 446.688,A -85,B 0,C 180,E1 -22933.526,E2 -22933.526} C_VEL
LIN {X 0,Y 223.928,Z 451.259,A -85,B 0,C 180,E1 -22936.635,E2 -22936.635} C_VEL
LIN {X 0,Y 231.528,Z 454.879,A -85,B 0,C 180,E1 -22939.506,E2 -22939.506} C_VEL
LIN {X 0,Y 236.982,Z 456.994,A -85,B 0,C 180,E1 -22941.473,E2 -22941.473} C_VEL
LIN {X 0,Y 241.993,Z 458.652,A -85,B 0,C 180,E1 -22943.329,E2 -22943.329} C_VEL
LIN {X 0,Y 246.816,Z 460.003,A -85,B 0,C 180,E1 -22945.27,E2 -22945.27} C_VEL
LIN {X 0,Y 249.835,Z 460.808,A -85,B 0,C 180,E1 -22946.775,E2 -22946.775} C_VEL
LIN {X 0,Y 253.06,Z 461.393,A -85,B 0,C 180,E1 -22948.786,E2 -22948.786} C_VEL
LIN {X 0,Y 254.353,Z 461.448,A -85,B 0,C 180,E1 -22950,E2 -22950} C_VEL
LIN {X 0,Y 252.4,Z 461.317,A -85,B 0,C 180,E1 -22951.596,E2 -22951.596} C_VEL
LIN {X 0,Y 249.801,Z 460.809,A -85,B 0,C 180,E1 -22953.226,E2 -22953.226} C_VEL
LIN {X 0,Y 246.367,Z 459.894,A -85,B 0,C 180,E1 -22954.909,E2 -22954.909} C_VEL
LIN {X 0,Y 240.811,Z 458.254,A -85,B 0,C 180,E1 -22957.132,E2 -22957.132} C_VEL
LIN {X 0,Y 234.984,Z 456.231,A -85,B 0,C 180,E1 -22959.263,E2 -22959.263} C_VEL
LIN {X 0,Y 225.964,Z 452.312,A -85,B 0,C 180,E1 -22962.575,E2 -22962.575} C_VEL
LIN {X 0,Y 218.755,Z 448.246,A -85,B 0,C 180,E1 -22965.464,E2 -22965.464} C_VEL
LIN {X 0,Y 211.511,Z 442.898,A -85,B 0,C 180,E1 -22968.747,E2 -22968.747} C_VEL
LIN {X 0,Y 205.215,Z 436.533,A -85,B 0,C 180,E1 -22972.13,E2 -22972.13} C_VEL
LIN {X 0,Y 201.088,Z 430.813,A -85,B 0,C 180,E1 -22974.796,E2 -22974.796} C_VEL
LIN {X 0,Y 197.558,Z 424.114,A -85,B 0,C 180,E1 -22977.546,E2 -22977.546} C_VEL
LIN {X 0,Y 194.936,Z 416.988,A -85,B 0,C 180,E1 -22980.089,E2 -22980.089} C_VEL
LIN {X 0,Y 192.901,Z 409.102,A -85,B 0,C 180,E1 -22982.519,E2 -22982.519} C_VEL
LIN {X 0,Y 190.534,Z 400.049,A -85,B 0,C 180,E1 -22985.044,E2 -22985.044} C_VEL
LIN {X 0,Y 187.327,Z 390.977,A -85,B 0,C 180,E1 -22987.528,E2 -22987.528} C_VEL
LIN {X 0,Y 182.849,Z 380.901,A -85,B 0,C 180,E1 -22990.3,E2 -22990.3} C_VEL
LIN {X 0,Y 178.375,Z 372.672,A -85,B 0,C 180,E1 -22992.69,E2 -22992.69} C_VEL
LIN {X 0,Y 176.024,Z 368.798,A -85,B 0,C 180,E1 -22993.851,E2 -22993.851} C_VEL
LIN {X 0,Y 173.927,Z 365.131,A -85,B 0,C 180,E1 -22994.948,E2 -22994.948} C_VEL
LIN {X 0,Y 172.114,Z 362.854,A -85,B 0,C 180,E1 -22995.768,E2 -22995.768} C_VEL
LIN {X 0,Y 171.422,Z 360.633,A -85,B 0,C 180,E1 -22996.244,E2 -22996.244} C_VEL
LIN {X 0,Y 171.425,Z 360.632,A -85,B 0,C 180,E1 -23001.165,E2 -23001.165} C_VEL
LIN {X 0,Y 171.405,Z 360.634,A -85,B 0,C 180,E1 -23005.089,E2 -23005.089} C_VEL
LIN {X 0,Y 171.447,Z 360.629,A -85,B 0,C 180,E1 -23010.536,E2 -23010.536} C_VEL
LIN {X 0,Y 171.443,Z 360.622,A -85,B 0,C 180,E1 -23015.801,E2 -23015.801} C_VEL
LIN {X 0,Y 171.576,Z 360.605,A -85,B 0,C 180,E1 -23020.873,E2 -23020.873} C_VEL
LIN {X 0,Y 171.593,Z 360.603,A -85,B 0,C 180,E1 -23025.776,E2 -23025.776} C_VEL
LIN {X 0,Y 171.873,Z 360.567,A -85,B 0,C 180,E1 -23030.588,E2 -23030.588} C_VEL
LIN {X 0,Y 171.821,Z 360.57,A -85,B 0,C 180,E1 -23035.309,E2 -23035.309} C_VEL
LIN {X 0,Y 172.331,Z 360.491,A -85,B 0,C 180,E1 -23040.001,E2 -23040.001} C_VEL
LIN {X 0,Y 171.822,Z 360.582,A -85,B 0,C 180,E1 -23044.694,E2 -23044.694} C_VEL
LIN {X 0,Y 171.889,Z 360.575,A -85,B 0,C 180,E1 -23049.414,E2 -23049.414} C_VEL
LIN {X 0,Y 171.572,Z 360.616,A -85,B 0,C 180,E1 -23054.229,E2 -23054.229} C_VEL
LIN {X 0,Y 171.54,Z 360.617,A -85,B 0,C 180,E1 -23059.558,E2 -23059.558} C_VEL
LIN {X 0,Y 171.455,Z 360.63,A -85,B 0,C 180,E1 -23061.65,E2 -23061.65} C_VEL
LIN {X 0,Y 171.583,Z 361.922,A -85,B 0,C 180,E1 -23066.781,E2 -23066.781} C_VEL
LIN {X 0,Y 171.8,Z 363.629,A -85,B 0,C 180,E1 -23072.129,E2 -23072.129} C_VEL
LIN {X 0,Y 171.98,Z 364.721,A -85,B 0,C 180,E1 -23075.185,E2 -23075.185} C_VEL
LIN {X 0,Y 172.197,Z 366.236,A -85,B 0,C 180,E1 -23079.154,E2 -23079.154} C_VEL
LIN {X 0,Y 172.316,Z 368.377,A -85,B 0,C 180,E1 -23084.207,E2 -23084.207} C_VEL
LIN {X 0,Y 173.324,Z 371.459,A -85,B 0,C 180,E1 -23084.812,E2 -23084.812} C_VEL
LIN {X 0,Y 174.779,Z 374.053,A -85,B 0,C 180,E1 -23085.561,E2 -23085.561} C_VEL
LIN {X 0,Y 178.416,Z 383.059,A -85,B 0,C 180,E1 -23087.697,E2 -23087.697} C_VEL
LIN {X 0,Y 181.647,Z 394.23,A -85,B 0,C 180,E1 -23090.249,E2 -23090.249} C_VEL
LIN {X 0,Y 183.537,Z 404.589,A -85,B 0,C 180,E1 -23092.615,E2 -23092.615} C_VEL
LIN {X 0,Y 184.477,Z 413.684,A -85,B 0,C 180,E1 -23094.802,E2 -23094.802} C_VEL
LIN {X 0,Y 184.706,Z 422.695,A -85,B 0,C 180,E1 -23097.142,E2 -23097.142} C_VEL
LIN {X 0,Y 184.397,Z 429.451,A -85,B 0,C 180,E1 -23099.034,E2 -23099.034} C_VEL
LIN {X 0,Y 183.833,Z 433.316,A -85,B 0,C 180,E1 -23100.199,E2 -23100.199} C_VEL
LIN {X 0,Y 180.613,Z 441.867,A -85,B 0,C 180,E1 -23102.793,E2 -23102.793} C_VEL
LIN {X 0,Y 177.644,Z 449.509,A -85,B 0,C 180,E1 -23105.721,E2 -23105.721} C_VEL
LIN {X 0,Y 174.943,Z 455.857,A -85,B 0,C 180,E1 -23108.804,E2 -23108.804} C_VEL
LIN {X 0,Y 172.596,Z 461.35,A -85,B 0,C 180,E1 -23112.218,E2 -23112.218} C_VEL
LIN {X 0,Y 170.836,Z 465.678,A -85,B 0,C 180,E1 -23115.71,E2 -23115.71} C_VEL
LIN {X 0,Y 170.056,Z 468.051,A -85,B 0,C 180,E1 -23118.075,E2 -23118.075} C_VEL
LIN {X 0,Y 169.077,Z 471.248,A -85,B 0,C 180,E1 -23122.837,E2 -23122.837} C_VEL
LIN {X 0,Y 168.933,Z 472.313,A -85,B 0,C 180,E1 -23125.227,E2 -23125.227} C_VEL
LIN {X 0,Y 168.87,Z 472.906,A -85,B 0,C 180,E1 -23127.615,E2 -23127.615} C_VEL
LIN {X 0,Y 168.972,Z 473.065,A -85,B 0,C 180,E1 -23130,E2 -23130} C_VEL
LIN {X 0,Y 168.853,Z 472.846,A -85,B 0,C 180,E1 -23132.627,E2 -23132.627} C_VEL
LIN {X 0,Y 168.868,Z 472.311,A -85,B 0,C 180,E1 -23134.775,E2 -23134.775} C_VEL
LIN {X 0,Y 169.435,Z 469.854,A -85,B 0,C 180,E1 -23139.55,E2 -23139.55} C_VEL
LIN {X 0,Y 170.433,Z 466.898,A -85,B 0,C 180,E1 -23143.109,E2 -23143.109} C_VEL
LIN {X 0,Y 171.889,Z 462.903,A -85,B 0,C 180,E1 -23146.631,E2 -23146.631} C_VEL
LIN {X 0,Y 174.153,Z 457.775,A -85,B 0,C 180,E1 -23150.061,E2 -23150.061} C_VEL
LIN {X 0,Y 176.421,Z 452.513,A -85,B 0,C 180,E1 -23152.855,E2 -23152.855} C_VEL
LIN {X 0,Y 178.14,Z 448.11,A -85,B 0,C 180,E1 -23154.849,E2 -23154.849} C_VEL
LIN {X 0,Y 180.568,Z 441.866,A -85,B 0,C 180,E1 -23157.215,E2 -23157.215} C_VEL
LIN {X 0,Y 183.797,Z 433.315,A -85,B 0,C 180,E1 -23159.808,E2 -23159.808} C_VEL
LIN {X 0,Y 184.553,Z 427.362,A -85,B 0,C 180,E1 -23161.575,E2 -23161.575} C_VEL
LIN {X 0,Y 184.689,Z 422.37,A -85,B 0,C 180,E1 -23162.953,E2 -23162.953} C_VEL
LIN {X 0,Y 184.051,Z 418.185,A -85,B 0,C 180,E1 -23164.234,E2 -23164.234} C_VEL
LIN {X 0,Y 181.264,Z 411.788,A -85,B 0,C 180,E1 -23166.446,E2 -23166.446} C_VEL
LIN {X 0,Y 178.62,Z 406.611,A -85,B 0,C 180,E1 -23168.211,E2 -23168.211} C_VEL
LIN {X 0,Y 176.68,Z 400.786,A -85,B 0,C 180,E1 -23169.859,E2 -23169.859} C_VEL
LIN {X 0,Y 174.312,Z 390.529,A -85,B 0,C 180,E1 -23172.383,E2 -23172.383} C_VEL
LIN {X 0,Y 171.359,Z 381.632,A -85,B 0,C 180,E1 -23174.654,E2 -23174.654} C_VEL
LIN {X 0,Y 169.516,Z 377.36,A -85,B 0,C 180,E1 -23175.784,E2 -23175.784} C_VEL
LIN {X 0,Y 167.582,Z 373.16,A -85,B 0,C 180,E1 -23176.98,E2 -23176.98} C_VEL
LIN {X 0,Y 165.75,Z 370.275,A -85,B 0,C 180,E1 -23177.966,E2 -23177.966} C_VEL
LIN {X 0,Y 165.187,Z 368.075,A -85,B 0,C 180,E1 -23178.378,E2 -23178.378} C_VEL
LIN {X 0,Y 165.161,Z 367.301,A -85,B 0,C 180,E1 -23180.334,E2 -23180.334} C_VEL
LIN {X 0,Y 164.958,Z 365.972,A -85,B 0,C 180,E1 -23184.046,E2 -23184.046} C_VEL
LIN {X 0,Y 164.744,Z 364.251,A -85,B 0,C 180,E1 -23189.207,E2 -23189.207} C_VEL
LIN {X 0,Y 164.554,Z 362.6,A -85,B 0,C 180,E1 -23194.715,E2 -23194.715} C_VEL
LIN {X 0,Y 164.485,Z 361.499,A -85,B 0,C 180,E1 -23200.05,E2 -23200.05} C_VEL
LIN {X 0,Y 164.502,Z 361.495,A -85,B 0,C 180,E1 -23205.146,E2 -23205.146} C_VEL
LIN {X 0,Y 164.803,Z 361.457,A -85,B 0,C 180,E1 -23210.177,E2 -23210.177} C_VEL
LIN {X 0,Y 164.851,Z 361.451,A -85,B 0,C 180,E1 -23212.651,E2 -23212.651} C_VEL
LIN {X 0,Y 165.05,Z 361.423,A -85,B 0,C 180,E1 -23217.558,E2 -23217.558} C_VEL
LIN {X 0,Y 165.294,Z 361.366,A -85,B 0,C 180,E1 -23219.999,E2 -23219.999} C_VEL
LIN {X 0,Y 164.77,Z 361.45,A -85,B 0,C 180,E1 -23224.892,E2 -23224.892} C_VEL
LIN {X 0,Y 164.846,Z 361.451,A -85,B 0,C 180,E1 -23227.347,E2 -23227.347} C_VEL
LIN {X 0,Y 164.75,Z 361.46,A -85,B 0,C 180,E1 -23231.145,E2 -23231.145} C_VEL
LIN {X 0,Y 164.484,Z 361.496,A -85,B 0,C 180,E1 -23237.402,E2 -23237.402} C_VEL
LIN {X 0,Y 164.471,Z 361.488,A -85,B 0,C 180,E1 -23239.988,E2 -23239.988} C_VEL
LIN {X 0,Y 164.384,Z 361.504,A -85,B 0,C 180,E1 -23246.127,E2 -23246.127} C_VEL
LIN {X 0,Y 164.374,Z 361.508,A -85,B 0,C 180,E1 -23251.227,E2 -23251.227} C_VEL
LIN {X 0,Y 164.345,Z 361.515,A -85,B 0,C 180,E1 -23256.774,E2 -23256.774} C_VEL
LIN {X 0,Y 164.406,Z 361.696,A -85,B 0,C 180,E1 -23261.292,E2 -23261.292} C_VEL
LIN {X 0,Y 165.388,Z 364.322,A -85,B 0,C 180,E1 -23261.907,E2 -23261.907} C_VEL
LIN {X 0,Y 167.542,Z 366.887,A -85,B 0,C 180,E1 -23263.009,E2 -23263.009} C_VEL
LIN {X 0,Y 169.381,Z 370.094,A -85,B 0,C 180,E1 -23264.077,E2 -23264.077} C_VEL
LIN {X 0,Y 170.404,Z 371.608,A -85,B 0,C 180,E1 -23264.62,E2 -23264.62} C_VEL
LIN {X 0,Y 174.863,Z 379.47,A -85,B 0,C 180,E1 -23267.178,E2 -23267.178} C_VEL
LIN {X 0,Y 178.769,Z 387.473,A -85,B 0,C 180,E1 -23269.634,E2 -23269.634} C_VEL
LIN {X 0,Y 182.248,Z 396.256,A -85,B 0,C 180,E1 -23272.232,E2 -23272.232} C_VEL
LIN {X 0,Y 185.09,Z 405.264,A -85,B 0,C 180,E1 -23274.912,E2 -23274.912} C_VEL
LIN {X 0,Y 187.09,Z 413.97,A -85,B 0,C 180,E1 -23277.582,E2 -23277.582} C_VEL
LIN {X 0,Y 188.943,Z 421.195,A -85,B 0,C 180,E1 -23280.051,E2 -23280.051} C_VEL
LIN {X 0,Y 191.51,Z 428.083,A -85,B 0,C 180,E1 -23282.763,E2 -23282.763} C_VEL
LIN {X 0,Y 195.91,Z 435.642,A -85,B 0,C 180,E1 -23286.276,E2 -23286.276} C_VEL
LIN {X 0,Y 201.024,Z 441.713,A -85,B 0,C 180,E1 -23289.537,E2 -23289.537} C_VEL
LIN {X 0,Y 206.448,Z 446.393,A -85,B 0,C 180,E1 -23292.395,E2 -23292.395} C_VEL
LIN {X 0,Y 213.845,Z 451.212,A -85,B 0,C 180,E1 -23295.783,E2 -23295.783} C_VEL
LIN {X 0,Y 222.033,Z 455.14,A -85,B 0,C 180,E1 -23299.052,E2 -23299.052} C_VEL
LIN {X 0,Y 227.62,Z 457.256,A -85,B 0,C 180,E1 -23301.119,E2 -23301.119} C_VEL
LIN {X 0,Y 233.52,Z 459.07,A -85,B 0,C 180,E1 -23303.289,E2 -23303.289} C_VEL
LIN {X 0,Y 239.629,Z 460.576,A -85,B 0,C 180,E1 -23305.677,E2 -23305.677} C_VEL
LIN {X 0,Y 241.78,Z 461.032,A -85,B 0,C 180,E1 -23306.667,E2 -23306.667} C_VEL
LIN {X 0,Y 246.007,Z 461.622,A -85,B 0,C 180,E1 -23309.076,E2 -23309.076} C_VEL
LIN {X 0,Y 247.032,Z 461.646,A -85,B 0,C 180,E1 -23310,E2 -23310} C_VEL
LIN {X 0,Y 244.744,Z 461.527,A -85,B 0,C 180,E1 -23311.646,E2 -23311.646} C_VEL
LIN {X 0,Y 241.763,Z 461.032,A -85,B 0,C 180,E1 -23313.333,E2 -23313.333} C_VEL
LIN {X 0,Y 237.769,Z 460.128,A -85,B 0,C 180,E1 -23315.087,E2 -23315.087} C_VEL
LIN {X 0,Y 232.957,Z 458.904,A -85,B 0,C 180,E1 -23316.931,E2 -23316.931} C_VEL
LIN {X 0,Y 224.823,Z 456.248,A -85,B 0,C 180,E1 -23319.9,E2 -23319.9} C_VEL
LIN {X 0,Y 216.447,Z 452.578,A -85,B 0,C 180,E1 -23323.137,E2 -23323.137} C_VEL
LIN {X 0,Y 208.681,Z 448.022,A -85,B 0,C 180,E1 -23326.503,E2 -23326.503} C_VEL
LIN {X 0,Y 201.896,Z 442.535,A -85,B 0,C 180,E1 -23329.974,E2 -23329.974} C_VEL
LIN {X 0,Y 196.758,Z 436.78,A -85,B 0,C 180,E1 -23333.136,E2 -23333.136} C_VEL
LIN {X 0,Y 192.558,Z 430.124,A -85,B 0,C 180,E1 -23336.318,E2 -23336.318} C_VEL
LIN {X 0,Y 189.596,Z 423.219,A -85,B 0,C 180,E1 -23339.174,E2 -23339.174} C_VEL
LIN {X 0,Y 187.319,Z 415.168,A -85,B 0,C 180,E1 -23342.03,E2 -23342.03} C_VEL
LIN {X 0,Y 185.465,Z 406.731,A -85,B 0,C 180,E1 -23344.639,E2 -23344.639} C_VEL
LIN {X 0,Y 182.963,Z 398.286,A -85,B 0,C 180,E1 -23347.154,E2 -23347.154} C_VEL
LIN {X 0,Y 180.241,Z 391.032,A -85,B 0,C 180,E1 -23349.312,E2 -23349.312} C_VEL
LIN {X 0,Y 176.647,Z 382.921,A -85,B 0,C 180,E1 -23351.759,E2 -23351.759} C_VEL
LIN {X 0,Y 171.333,Z 373.31,A -85,B 0,C 180,E1 -23354.858,E2 -23354.858} C_VEL
LIN {X 0,Y 169.251,Z 369.916,A -85,B 0,C 180,E1 -23355.991,E2 -23355.991} C_VEL
LIN {X 0,Y 167.442,Z 366.677,A -85,B 0,C 180,E1 -23357.055,E2 -23357.055} C_VEL
LIN {X 0,Y 165.158,Z 363.947,A -85,B 0,C 180,E1 -23358.226,E2 -23358.226} C_VEL
LIN {X 0,Y 164.389,Z 361.508,A -85,B 0,C 180,E1 -23358.805,E2 -23358.805} C_VEL
LIN {X 0,Y 164.343,Z 361.512,A -85,B 0,C 180,E1 -23364.343,E2 -23364.343} C_VEL
LIN {X 0,Y 164.389,Z 361.506,A -85,B 0,C 180,E1 -23369.136,E2 -23369.136} C_VEL
LIN {X 0,Y 164.405,Z 361.497,A -85,B 0,C 180,E1 -23374.694,E2 -23374.694} C_VEL
LIN {X 0,Y 164.483,Z 361.487,A -85,B 0,C 180,E1 -23380.053,E2 -23380.053} C_VEL
LIN {X 0,Y 164.535,Z 361.481,A -85,B 0,C 180,E1 -23385.152,E2 -23385.152} C_VEL
LIN {X 0,Y 164.797,Z 361.448,A -85,B 0,C 180,E1 -23390.18,E2 -23390.18} C_VEL
LIN {X 0,Y 164.846,Z 361.451,A -85,B 0,C 180,E1 -23392.653,E2 -23392.653} C_VEL
LIN {X 0,Y 165.049,Z 361.388,A -85,B 0,C 180,E1 -23397.561,E2 -23397.561} C_VEL
LIN {X 0,Y 165.294,Z 361.366,A -85,B 0,C 180,E1 -23400.001,E2 -23400.001} C_VEL
LIN {X 0,Y 164.772,Z 361.46,A -85,B 0,C 180,E1 -23404.895,E2 -23404.895} C_VEL
LIN {X 0,Y 164.851,Z 361.452,A -85,B 0,C 180,E1 -23407.349,E2 -23407.349} C_VEL
LIN {X 0,Y 164.743,Z 361.466,A -85,B 0,C 180,E1 -23411.132,E2 -23411.132} C_VEL
LIN {X 0,Y 164.479,Z 361.499,A -85,B 0,C 180,E1 -23417.405,E2 -23417.405} C_VEL
LIN {X 0,Y 164.474,Z 361.498,A -85,B 0,C 180,E1 -23419.99,E2 -23419.99} C_VEL
LIN {X 0,Y 164.557,Z 362.583,A -85,B 0,C 180,E1 -23425.284,E2 -23425.284} C_VEL
LIN {X 0,Y 164.75,Z 364.459,A -85,B 0,C 180,E1 -23431.442,E2 -23431.442} C_VEL
LIN {X 0,Y 164.986,Z 366.203,A -85,B 0,C 180,E1 -23436.612,E2 -23436.612} C_VEL
LIN {X 0,Y 165.204,Z 368.098,A -85,B 0,C 180,E1 -23441.52,E2 -23441.52} C_VEL
LIN {X 0,Y 165.349,Z 368.969,A -85,B 0,C 180,E1 -23441.767,E2 -23441.767} C_VEL
LIN {X 0,Y 166.63,Z 371.906,A -85,B 0,C 180,E1 -23442.519,E2 -23442.519} C_VEL
LIN {X 0,Y 168.006,Z 373.934,A -85,B 0,C 180,E1 -23443.268,E2 -23443.268} C_VEL
LIN {X 0,Y 169.86,Z 377.921,A -85,B 0,C 180,E1 -23444.401,E2 -23444.401} C_VEL
LIN {X 0,Y 173.38,Z 387.367,A -85,B 0,C 180,E1 -23446.857,E2 -23446.857} C_VEL
LIN {X 0,Y 175.579,Z 395.613,A -85,B 0,C 180,E1 -23448.882,E2 -23448.882} C_VEL
LIN {X 0,Y 177.16,Z 404.079,A -85,B 0,C 180,E1 -23450.959,E2 -23450.959} C_VEL
LIN {X 0,Y 178.122,Z 413.468,A -85,B 0,C 180,E1 -23453.347,E2 -23453.347} C_VEL
LIN {X 0,Y 178.31,Z 422.689,A -85,B 0,C 180,E1 -23455.866,E2 -23455.866} C_VEL
LIN {X 0,Y 178.015,Z 429.245,A -85,B 0,C 180,E1 -23457.793,E2 -23457.793} C_VEL
LIN {X 0,Y 177.522,Z 433.114,A -85,B 0,C 180,E1 -23459.025,E2 -23459.025} C_VEL
LIN {X 0,Y 175.634,Z 438.418,A -85,B 0,C 180,E1 -23460.647,E2 -23460.647} C_VEL
LIN {X 0,Y 173.071,Z 444.619,A -85,B 0,C 180,E1 -23462.817,E2 -23462.817} C_VEL
LIN {X 0,Y 170.92,Z 449.87,A -85,B 0,C 180,E1 -23464.998,E2 -23464.998} C_VEL
LIN {X 0,Y 168.314,Z 455.66,A -85,B 0,C 180,E1 -23467.927,E2 -23467.927} C_VEL
LIN {X 0,Y 165.837,Z 461.154,A -85,B 0,C 180,E1 -23471.468,E2 -23471.468} C_VEL
LIN {X 0,Y 163.913,Z 465.481,A -85,B 0,C 180,E1 -23475.093,E2 -23475.093} C_VEL
LIN {X 0,Y 163.099,Z 467.854,A -85,B 0,C 180,E1 -23477.558,E2 -23477.558} C_VEL
LIN {X 0,Y 162.416,Z 469.658,A -85,B 0,C 180,E1 -23480.033,E2 -23480.033} C_VEL
LIN {X 0,Y 161.852,Z 472.117,A -85,B 0,C 180,E1 -23485.018,E2 -23485.018} C_VEL
LIN {X 0,Y 161.8,Z 472.711,A -85,B 0,C 180,E1 -23487.511,E2 -23487.511} C_VEL
LIN {X 0,Y 161.884,Z 472.87,A -85,B 0,C 180,E1 -23490,E2 -23490} C_VEL
LIN {X 0,Y 161.763,Z 472.71,A -85,B 0,C 180,E1 -23492.49,E2 -23492.49} C_VEL
LIN {X 0,Y 161.795,Z 472.115,A -85,B 0,C 180,E1 -23494.984,E2 -23494.984} C_VEL
LIN {X 0,Y 162.416,Z 469.658,A -85,B 0,C 180,E1 -23499.967,E2 -23499.967} C_VEL
LIN {X 0,Y 163.477,Z 466.701,A -85,B 0,C 180,E1 -23503.677,E2 -23503.677} C_VEL
LIN {X 0,Y 165.08,Z 462.707,A -85,B 0,C 180,E1 -23507.338,E2 -23507.338} C_VEL
LIN {X 0,Y 167.459,Z 457.577,A -85,B 0,C 180,E1 -23510.9,E2 -23510.9} C_VEL
LIN {X 0,Y 169.882,Z 452.317,A -85,B 0,C 180,E1 -23513.788,E2 -23513.788} C_VEL
LIN {X 0,Y 172.485,Z 445.995,A -85,B 0,C 180,E1 -23516.628,E2 -23516.628} C_VEL
LIN {X 0,Y 174.903,Z 440.043,A -85,B 0,C 180,E1 -23518.828,E2 -23518.828} C_VEL
LIN {X 0,Y 176.988,Z 435.039,A -85,B 0,C 180,E1 -23520.417,E2 -23520.417} C_VEL
LIN {X 0,Y 177.799,Z 431.181,A -85,B 0,C 180,E1 -23521.584,E2 -23521.584} C_VEL
LIN {X 0,Y 178.249,Z 423.678,A -85,B 0,C 180,E1 -23523.854,E2 -23523.854} C_VEL
LIN {X 0,Y 178.222,Z 416.251,A -85,B 0,C 180,E1 -23525.916,E2 -23525.916} C_VEL
LIN {X 0,Y 177.591,Z 407.465,A -85,B 0,C 180,E1 -23528.187,E2 -23528.187} C_VEL
LIN {X 0,Y 176.68,Z 400.786,A -85,B 0,C 180,E1 -23529.859,E2 -23529.859} C_VEL
LIN {X 0,Y 175.239,Z 396.446,A -85,B 0,C 180,E1 -23531.077,E2 -23531.077} C_VEL
LIN {X 0,Y 173.063,Z 392.681,A -85,B 0,C 180,E1 -23532.41,E2 -23532.41} C_VEL
LIN {X 0,Y 167.781,Z 385.899,A -85,B 0,C 180,E1 -23535.248,E2 -23535.248} C_VEL
LIN {X 0,Y 164.469,Z 380.981,A -85,B 0,C 180,E1 -23537.129,E2 -23537.129} C_VEL
LIN {X 0,Y 162.919,Z 377.719,A -85,B 0,C 180,E1 -23538.14,E2 -23538.14} C_VEL
LIN {X 0,Y 161.144,Z 374.026,A -85,B 0,C 180,E1 -23539.339,E2 -23539.339} C_VEL
LIN {X 0,Y 160.519,Z 372.918,A -85,B 0,C 180,E1 -23539.748,E2 -23539.748} C_VEL
LIN {X 0,Y 158.627,Z 369.972,A -85,B 0,C 180,E1 -23540.906,E2 -23540.906} C_VEL
LIN {X 0,Y 158.003,Z 367.764,A -85,B 0,C 180,E1 -23541.483,E2 -23541.483} C_VEL
LIN {X 0,Y 157.861,Z 366.703,A -85,B 0,C 180,E1 -23544.635,E2 -23544.635} C_VEL
LIN {X 0,Y 157.736,Z 365.683,A -85,B 0,C 180,E1 -23547.838,E2 -23547.838} C_VEL
LIN {X 0,Y 157.541,Z 364.035,A -85,B 0,C 180,E1 -23553.504,E2 -23553.504} C_VEL
LIN {X 0,Y 157.424,Z 362.499,A -85,B 0,C 180,E1 -23559.638,E2 -23559.638} C_VEL
LIN {X 0,Y 157.438,Z 362.375,A -85,B 0,C 180,E1 -23564.463,E2 -23564.463} C_VEL
LIN {X 0,Y 157.727,Z 362.339,A -85,B 0,C 180,E1 -23569.732,E2 -23569.732} C_VEL
LIN {X 0,Y 157.808,Z 362.328,A -85,B 0,C 180,E1 -23572.321,E2 -23572.321} C_VEL
LIN {X 0,Y 158.257,Z 362.241,A -85,B 0,C 180,E1 -23579.999,E2 -23579.999} C_VEL
LIN {X 0,Y 157.803,Z 362.327,A -85,B 0,C 180,E1 -23587.677,E2 -23587.677} C_VEL
LIN {X 0,Y 157.68,Z 362.342,A -85,B 0,C 180,E1 -23591.314,E2 -23591.314} C_VEL
LIN {X 0,Y 157.461,Z 362.364,A -85,B 0,C 180,E1 -23595.532,E2 -23595.532} C_VEL
LIN {X 0,Y 157.366,Z 362.376,A -85,B 0,C 180,E1 -23600.932,E2 -23600.932} C_VEL
LIN {X 0,Y 157.308,Z 362.388,A -85,B 0,C 180,E1 -23606.68,E2 -23606.68} C_VEL
LIN {X 0,Y 157.276,Z 362.395,A -85,B 0,C 180,E1 -23612.426,E2 -23612.426} C_VEL
LIN {X 0,Y 157.29,Z 362.392,A -85,B 0,C 180,E1 -23617.473,E2 -23617.473} C_VEL
LIN {X 0,Y 157.274,Z 362.393,A -85,B 0,C 180,E1 -23618.255,E2 -23618.255} C_VEL
LIN {X 0,Y 158.096,Z 364.895,A -85,B 0,C 180,E1 -23618.897,E2 -23618.897} C_VEL
LIN {X 0,Y 159.955,Z 367.07,A -85,B 0,C 180,E1 -23619.991,E2 -23619.991} C_VEL
LIN {X 0,Y 160.663,Z 367.889,A -85,B 0,C 180,E1 -23620.41,E2 -23620.41} C_VEL
LIN {X 0,Y 162.458,Z 371.059,A -85,B 0,C 180,E1 -23621.587,E2 -23621.587} C_VEL
LIN {X 0,Y 163.724,Z 372.856,A -85,B 0,C 180,E1 -23622.328,E2 -23622.328} C_VEL
LIN {X 0,Y 165.856,Z 376.136,A -85,B 0,C 180,E1 -23623.592,E2 -23623.592} C_VEL
LIN {X 0,Y 171.131,Z 386.24,A -85,B 0,C 180,E1 -23627.119,E2 -23627.119} C_VEL
LIN {X 0,Y 175.327,Z 396.28,A -85,B 0,C 180,E1 -23630.408,E2 -23630.408} C_VEL
LIN {X 0,Y 178.175,Z 405.278,A -85,B 0,C 180,E1 -23633.279,E2 -23633.279} C_VEL
LIN {X 0,Y 180.051,Z 412.784,A -85,B 0,C 180,E1 -23635.722,E2 -23635.722} C_VEL
LIN {X 0,Y 181.778,Z 421.418,A -85,B 0,C 180,E1 -23638.741,E2 -23638.741} C_VEL
LIN {X 0,Y 184.538,Z 429.831,A -85,B 0,C 180,E1 -23642.237,E2 -23642.237} C_VEL
LIN {X 0,Y 187.641,Z 435.755,A -85,B 0,C 180,E1 -23645.104,E2 -23645.104} C_VEL
LIN {X 0,Y 192.36,Z 441.964,A -85,B 0,C 180,E1 -23648.571,E2 -23648.571} C_VEL
LIN {X 0,Y 196.839,Z 446.231,A -85,B 0,C 180,E1 -23651.256,E2 -23651.256} C_VEL
LIN {X 0,Y 203.859,Z 451.174,A -85,B 0,C 180,E1 -23654.856,E2 -23654.856} C_VEL
LIN {X 0,Y 212.479,Z 455.404,A -85,B 0,C 180,E1 -23658.553,E2 -23658.553} C_VEL
LIN {X 0,Y 220.266,Z 458.178,A -85,B 0,C 180,E1 -23661.529,E2 -23661.529} C_VEL
LIN {X 0,Y 226.246,Z 459.824,A -85,B 0,C 180,E1 -23663.727,E2 -23663.727} C_VEL
LIN {X 0,Y 233.537,Z 461.262,A -85,B 0,C 180,E1 -23666.549,E2 -23666.549} C_VEL
LIN {X 0,Y 236.999,Z 461.74,A -85,B 0,C 180,E1 -23668.301,E2 -23668.301} C_VEL
LIN {X 0,Y 238.96,Z 461.855,A -85,B 0,C 180,E1 -23669.424,E2 -23669.424} C_VEL
LIN {X 0,Y 239.679,Z 461.845,A -85,B 0,C 180,E1 -23670,E2 -23670} C_VEL
LIN {X 0,Y 236.923,Z 461.742,A -85,B 0,C 180,E1 -23671.7,E2 -23671.7} C_VEL
LIN {X 0,Y 233.546,Z 461.261,A -85,B 0,C 180,E1 -23673.45,E2 -23673.45} C_VEL
LIN {X 0,Y 226.248,Z 459.822,A -85,B 0,C 180,E1 -23676.277,E2 -23676.277} C_VEL
LIN {X 0,Y 218.089,Z 457.523,A -85,B 0,C 180,E1 -23679.272,E2 -23679.272} C_VEL
LIN {X 0,Y 209.053,Z 453.918,A -85,B 0,C 180,E1 -23682.862,E2 -23682.862} C_VEL
LIN {X 0,Y 201.669,Z 449.841,A -85,B 0,C 180,E1 -23686.188,E2 -23686.188} C_VEL
LIN {X 0,Y 194.517,Z 444.206,A -85,B 0,C 180,E1 -23690.054,E2 -23690.054} C_VEL
LIN {X 0,Y 189.068,Z 437.891,A -85,B 0,C 180,E1 -23693.752,E2 -23693.752} C_VEL
LIN {X 0,Y 185.235,Z 431.286,A -85,B 0,C 180,E1 -23697.084,E2 -23697.084} C_VEL
LIN {X 0,Y 182.67,Z 424.569,A -85,B 0,C 180,E1 -23700.01,E2 -23700.01} C_VEL
LIN {X 0,Y 180.715,Z 416.592,A -85,B 0,C 180,E1 -23702.988,E2 -23702.988} C_VEL
LIN {X 0,Y 179.168,Z 408.943,A -85,B 0,C 180,E1 -23705.52,E2 -23705.52} C_VEL
LIN {X 0,Y 176.734,Z 400.497,A -85,B 0,C 180,E1 -23708.247,E2 -23708.247} C_VEL
LIN {X 0,Y 173.918,Z 392.803,A -85,B 0,C 180,E1 -23710.742,E2 -23710.742} C_VEL
LIN {X 0,Y 170.027,Z 384.1,A -85,B 0,C 180,E1 -23713.633,E2 -23713.633} C_VEL
LIN {X 0,Y 165.849,Z 376.168,A -85,B 0,C 180,E1 -23716.406,E2 -23716.406} C_VEL
LIN {X 0,Y 163.517,Z 372.398,A -85,B 0,C 180,E1 -23717.814,E2 -23717.814} C_VEL
LIN {X 0,Y 160.856,Z 368.49,A -85,B 0,C 180,E1 -23719.425,E2 -23719.425} C_VEL
LIN {X 0,Y 160.198,Z 367.256,A -85,B 0,C 180,E1 -23719.878,E2 -23719.878} C_VEL
LIN {X 0,Y 158.097,Z 364.916,A -85,B 0,C 180,E1 -23721.103,E2 -23721.103} C_VEL
LIN {X 0,Y 157.267,Z 362.394,A -85,B 0,C 180,E1 -23721.822,E2 -23721.822} C_VEL
LIN {X 0,Y 157.29,Z 362.391,A -85,B 0,C 180,E1 -23724.491,E2 -23724.491} C_VEL
LIN {X 0,Y 157.293,Z 362.392,A -85,B 0,C 180,E1 -23728.096,E2 -23728.096} C_VEL
LIN {X 0,Y 157.314,Z 362.387,A -85,B 0,C 180,E1 -23733.466,E2 -23733.466} C_VEL
LIN {X 0,Y 157.391,Z 362.37,A -85,B 0,C 180,E1 -23739.671,E2 -23739.671} C_VEL
LIN {X 0,Y 157.461,Z 362.364,A -85,B 0,C 180,E1 -23744.468,E2 -23744.468} C_VEL
LIN {X 0,Y 157.726,Z 362.33,A -85,B 0,C 180,E1 -23749.735,E2 -23749.735} C_VEL
LIN {X 0,Y 157.803,Z 362.327,A -85,B 0,C 180,E1 -23752.323,E2 -23752.323} C_VEL
LIN {X 0,Y 158.257,Z 362.241,A -85,B 0,C 180,E1 -23760.001,E2 -23760.001} C_VEL
LIN {X 0,Y 157.808,Z 362.329,A -85,B 0,C 180,E1 -23767.679,E2 -23767.679} C_VEL
LIN {X 0,Y 157.673,Z 362.347,A -85,B 0,C 180,E1 -23771.302,E2 -23771.302} C_VEL
LIN {X 0,Y 157.438,Z 362.377,A -85,B 0,C 180,E1 -23775.537,E2 -23775.537} C_VEL
LIN {X 0,Y 157.424,Z 362.496,A -85,B 0,C 180,E1 -23780.362,E2 -23780.362} C_VEL
LIN {X 0,Y 157.563,Z 364.029,A -85,B 0,C 180,E1 -23786.492,E2 -23786.492} C_VEL
LIN {X 0,Y 157.739,Z 365.733,A -85,B 0,C 180,E1 -23792.322,E2 -23792.322} C_VEL
LIN {X 0,Y 157.949,Z 367.17,A -85,B 0,C 180,E1 -23796.783,E2 -23796.783} C_VEL
LIN {X 0,Y 158.047,Z 367.989,A -85,B 0,C 180,E1 -23798.642,E2 -23798.642} C_VEL
LIN {X 0,Y 158.997,Z 370.75,A -85,B 0,C 180,E1 -23799.332,E2 -23799.332} C_VEL
LIN {X 0,Y 161.088,Z 373.829,A -85,B 0,C 180,E1 -23800.611,E2 -23800.611} C_VEL
LIN {X 0,Y 162.807,Z 377.526,A -85,B 0,C 180,E1 -23801.792,E2 -23801.792} C_VEL
LIN {X 0,Y 163.894,Z 379.659,A -85,B 0,C 180,E1 -23802.485,E2 -23802.485} C_VEL
LIN {X 0,Y 166.247,Z 385.419,A -85,B 0,C 180,E1 -23804.229,E2 -23804.229} C_VEL
LIN {X 0,Y 168.764,Z 393.151,A -85,B 0,C 180,E1 -23806.385,E2 -23806.385} C_VEL
LIN {X 0,Y 170.822,Z 403.236,A -85,B 0,C 180,E1 -23809.068,E2 -23809.068} C_VEL
LIN {X 0,Y 171.79,Z 413.248,A -85,B 0,C 180,E1 -23811.76,E2 -23811.76} C_VEL
LIN {X 0,Y 172.01,Z 422.361,A -85,B 0,C 180,E1 -23814.394,E2 -23814.394} C_VEL
LIN {X 0,Y 171.471,Z 430.977,A -85,B 0,C 180,E1 -23817.108,E2 -23817.108} C_VEL
LIN {X 0,Y 170.829,Z 434.84,A -85,B 0,C 180,E1 -23818.363,E2 -23818.363} C_VEL
LIN {X 0,Y 166.756,Z 444.422,A -85,B 0,C 180,E1 -23821.697,E2 -23821.697} C_VEL
LIN {X 0,Y 163.878,Z 450.963,A -85,B 0,C 180,E1 -23824.605,E2 -23824.605} C_VEL
LIN {X 0,Y 161.739,Z 455.464,A -85,B 0,C 180,E1 -23826.979,E2 -23826.979} C_VEL
LIN {X 0,Y 159.083,Z 460.957,A -85,B 0,C 180,E1 -23830.65,E2 -23830.65} C_VEL
LIN {X 0,Y 157.016,Z 465.284,A -85,B 0,C 180,E1 -23834.422,E2 -23834.422} C_VEL
LIN {X 0,Y 156.124,Z 467.657,A -85,B 0,C 180,E1 -23836.993,E2 -23836.993} C_VEL
LIN {X 0,Y 155.419,Z 469.461,A -85,B 0,C 180,E1 -23839.579,E2 -23839.579} C_VEL
LIN {X 0,Y 154.755,Z 471.92,A -85,B 0,C 180,E1 -23844.789,E2 -23844.789} C_VEL
LIN {X 0,Y 154.715,Z 472.636,A -85,B 0,C 180,E1 -23847.983,E2 -23847.983} C_VEL
LIN {X 0,Y 154.687,Z 472.666,A -85,B 0,C 180,E1 -23851.695,E2 -23851.695} C_VEL
LIN {X 0,Y 154.715,Z 471.919,A -85,B 0,C 180,E1 -23855.213,E2 -23855.213} C_VEL
LIN {X 0,Y 155.419,Z 469.461,A -85,B 0,C 180,E1 -23860.421,E2 -23860.421} C_VEL
LIN {X 0,Y 156.546,Z 466.504,A -85,B 0,C 180,E1 -23864.295,E2 -23864.295} C_VEL
LIN {X 0,Y 158.305,Z 462.51,A -85,B 0,C 180,E1 -23868.105,E2 -23868.105} C_VEL
LIN {X 0,Y 160.796,Z 457.38,A -85,B 0,C 180,E1 -23871.809,E2 -23871.809} C_VEL
LIN {X 0,Y 163.378,Z 452.12,A -85,B 0,C 180,E1 -23874.797,E2 -23874.797} C_VEL
LIN {X 0,Y 165.438,Z 447.412,A -85,B 0,C 180,E1 -23877.055,E2 -23877.055} C_VEL
LIN {X 0,Y 168.028,Z 441.473,A -85,B 0,C 180,E1 -23879.436,E2 -23879.436} C_VEL
LIN {X 0,Y 170.815,Z 434.84,A -85,B 0,C 180,E1 -23881.64,E2 -23881.64} C_VEL
LIN {X 0,Y 171.756,Z 428.043,A -85,B 0,C 180,E1 -23883.884,E2 -23883.884} C_VEL
LIN {X 0,Y 172.04,Z 418.78,A -85,B 0,C 180,E1 -23886.686,E2 -23886.686} C_VEL
LIN {X 0,Y 171.524,Z 409.237,A -85,B 0,C 180,E1 -23889.34,E2 -23889.34} C_VEL
LIN {X 0,Y 170.429,Z 400.772,A -85,B 0,C 180,E1 -23891.598,E2 -23891.598} C_VEL
LIN {X 0,Y 167.739,Z 389.596,A -85,B 0,C 180,E1 -23894.578,E2 -23894.578} C_VEL
LIN {X 0,Y 164.528,Z 381.088,A -85,B 0,C 180,E1 -23897.093,E2 -23897.093} C_VEL
LIN {X 0,Y 164.469,Z 380.981,A -85,B 0,C 180,E1 -23897.129,E2 -23897.129} C_VEL
LIN {X 0,Y 162.071,Z 378.116,A -85,B 0,C 180,E1 -23898.43,E2 -23898.43} C_VEL
LIN {X 0,Y 159.17,Z 376.209,A -85,B 0,C 180,E1 -23899.869,E2 -23899.869} C_VEL
LIN {X 0,Y 153.398,Z 372.727,A -85,B 0,C 180,E1 -23902.982,E2 -23902.982} C_VEL
LIN {X 0,Y 151.474,Z 369.841,A -85,B 0,C 180,E1 -23904.346,E2 -23904.346} C_VEL
LIN {X 0,Y 150.808,Z 367.508,A -85,B 0,C 180,E1 -23904.983,E2 -23904.983} C_VEL
LIN {X 0,Y 150.599,Z 366.295,A -85,B 0,C 180,E1 -23909.112,E2 -23909.112} C_VEL
LIN {X 0,Y 150.509,Z 365.356,A -85,B 0,C 180,E1 -23912.524,E2 -23912.524} C_VEL
LIN {X 0,Y 150.388,Z 363.994,A -85,B 0,C 180,E1 -23918.045,E2 -23918.045} C_VEL
LIN {X 0,Y 150.37,Z 363.367,A -85,B 0,C 180,E1 -23920.902,E2 -23920.902} C_VEL
LIN {X 0,Y 150.437,Z 363.247,A -85,B 0,C 180,E1 -23926.49,E2 -23926.49} C_VEL
LIN {X 0,Y 150.649,Z 363.22,A -85,B 0,C 180,E1 -23929.244,E2 -23929.244} C_VEL
LIN {X 0,Y 150.743,Z 363.209,A -85,B 0,C 180,E1 -23931.958,E2 -23931.958} C_VEL
LIN {X 0,Y 151.217,Z 363.116,A -85,B 0,C 180,E1 -23939.999,E2 -23939.999} C_VEL
LIN {X 0,Y 150.739,Z 363.205,A -85,B 0,C 180,E1 -23948.039,E2 -23948.039} C_VEL
LIN {X 0,Y 150.61,Z 363.224,A -85,B 0,C 180,E1 -23951.499,E2 -23951.499} C_VEL
LIN {X 0,Y 150.367,Z 363.252,A -85,B 0,C 180,E1 -23956.285,E2 -23956.285} C_VEL
LIN {X 0,Y 150.348,Z 363.249,A -85,B 0,C 180,E1 -23960.789,E2 -23960.789} C_VEL
LIN {X 0,Y 150.239,Z 363.271,A -85,B 0,C 180,E1 -23967.278,E2 -23967.278} C_VEL
LIN {X 0,Y 150.216,Z 363.273,A -85,B 0,C 180,E1 -23972.633,E2 -23972.633} C_VEL
LIN {X 0,Y 150.215,Z 363.274,A -85,B 0,C 180,E1 -23974.763,E2 -23974.763} C_VEL
LIN {X 0,Y 151.09,Z 365.831,A -85,B 0,C 180,E1 -23975.55,E2 -23975.55} C_VEL
LIN {X 0,Y 153.324,Z 368.253,A -85,B 0,C 180,E1 -23977.079,E2 -23977.079} C_VEL
LIN {X 0,Y 154.185,Z 369.953,A -85,B 0,C 180,E1 -23977.769,E2 -23977.769} C_VEL
LIN {X 0,Y 156.323,Z 372.861,A -85,B 0,C 180,E1 -23979.213,E2 -23979.213} C_VEL
LIN {X 0,Y 161.786,Z 381.997,A -85,B 0,C 180,E1 -23983.084,E2 -23983.084} C_VEL
LIN {X 0,Y 165.747,Z 389.989,A -85,B 0,C 180,E1 -23986.121,E2 -23986.121} C_VEL
LIN {X 0,Y 169.08,Z 398.243,A -85,B 0,C 180,E1 -23989.061,E2 -23989.061} C_VEL
LIN {X 0,Y 171.498,Z 405.946,A -85,B 0,C 180,E1 -23991.719,E2 -23991.719} C_VEL
LIN {X 0,Y 173.509,Z 414.133,A -85,B 0,C 180,E1 -23994.6,E2 -23994.6} C_VEL
LIN {X 0,Y 175.161,Z 423.472,A -85,B 0,C 180,E1 -23998.084,E2 -23998.084} C_VEL
LIN {X 0,Y 177.016,Z 429.845,A -85,B 0,C 180,E1 -24000.86,E2 -24000.86} C_VEL
LIN {X 0,Y 179.784,Z 436.208,A -85,B 0,C 180,E1 -24004.037,E2 -24004.037} C_VEL
LIN {X 0,Y 183.897,Z 442.21,A -85,B 0,C 180,E1 -24007.532,E2 -24007.532} C_VEL
LIN {X 0,Y 189.329,Z 447.677,A -85,B 0,C 180,E1 -24011.218,E2 -24011.218} C_VEL
LIN {X 0,Y 196.406,Z 452.491,A -85,B 0,C 180,E1 -24015.043,E2 -24015.043} C_VEL
LIN {X 0,Y 202.949,Z 455.667,A -85,B 0,C 180,E1 -24018.008,E2 -24018.008} C_VEL
LIN {X 0,Y 208.566,Z 457.789,A -85,B 0,C 180,E1 -24020.3,E2 -24020.3} C_VEL
LIN {X 0,Y 214.209,Z 459.424,A -85,B 0,C 180,E1 -24022.459,E2 -24022.459} C_VEL
LIN {X 0,Y 219.726,Z 460.621,A -85,B 0,C 180,E1 -24024.494,E2 -24024.494} C_VEL
LIN {X 0,Y 225.287,Z 461.563,A -85,B 0,C 180,E1 -24026.607,E2 -24026.607} C_VEL
LIN {X 0,Y 228.957,Z 461.96,A -85,B 0,C 180,E1 -24028.241,E2 -24028.241} C_VEL
LIN {X 0,Y 232.176,Z 462.048,A -85,B 0,C 180,E1 -24030,E2 -24030} C_VEL
LIN {X 0,Y 228.925,Z 461.961,A -85,B 0,C 180,E1 -24031.759,E2 -24031.759} C_VEL
LIN {X 0,Y 224.839,Z 461.503,A -85,B 0,C 180,E1 -24033.584,E2 -24033.584} C_VEL
LIN {X 0,Y 218.98,Z 460.476,A -85,B 0,C 180,E1 -24035.788,E2 -24035.788} C_VEL
LIN {X 0,Y 212.918,Z 459.064,A -85,B 0,C 180,E1 -24038.019,E2 -24038.019} C_VEL
LIN {X 0,Y 207.121,Z 457.307,A -85,B 0,C 180,E1 -24040.263,E2 -24040.263} C_VEL
LIN {X 0,Y 197.506,Z 453.107,A -85,B 0,C 180,E1 -24044.423,E2 -24044.423} C_VEL
LIN {X 0,Y 191.574,Z 449.425,A -85,B 0,C 180,E1 -24047.484,E2 -24047.484} C_VEL
LIN {X 0,Y 186.119,Z 444.753,A -85,B 0,C 180,E1 -24050.845,E2 -24050.845} C_VEL
LIN {X 0,Y 181.21,Z 438.587,A -85,B 0,C 180,E1 -24054.64,E2 -24054.64} C_VEL
LIN {X 0,Y 178.285,Z 433.094,A -85,B 0,C 180,E1 -24057.592,E2 -24057.592} C_VEL
LIN {X 0,Y 176.019,Z 426.613,A -85,B 0,C 180,E1 -24060.618,E2 -24060.618} C_VEL
LIN {X 0,Y 174.131,Z 417.824,A -85,B 0,C 180,E1 -24064.086,E2 -24064.086} C_VEL
LIN {X 0,Y 172.552,Z 409.766,A -85,B 0,C 180,E1 -24066.939,E2 -24066.939} C_VEL
LIN {X 0,Y 169.975,Z 400.845,A -85,B 0,C 180,E1 -24070.041,E2 -24070.041} C_VEL
LIN {X 0,Y 166.487,Z 391.717,A -85,B 0,C 180,E1 -24073.267,E2 -24073.267} C_VEL
LIN {X 0,Y 162.673,Z 383.723,A -85,B 0,C 180,E1 -24076.273,E2 -24076.273} C_VEL
LIN {X 0,Y 158.619,Z 376.62,A -85,B 0,C 180,E1 -24079.193,E2 -24079.193} C_VEL
LIN {X 0,Y 156.095,Z 372.618,A -85,B 0,C 180,E1 -24080.927,E2 -24080.927} C_VEL
LIN {X 0,Y 154.054,Z 369.687,A -85,B 0,C 180,E1 -24082.336,E2 -24082.336} C_VEL
LIN {X 0,Y 153.32,Z 368.272,A -85,B 0,C 180,E1 -24082.92,E2 -24082.92} C_VEL
LIN {X 0,Y 151.09,Z 365.831,A -85,B 0,C 180,E1 -24084.45,E2 -24084.45} C_VEL
LIN {X 0,Y 150.219,Z 363.274,A -85,B 0,C 180,E1 -24085.34,E2 -24085.34} C_VEL
LIN {X 0,Y 150.206,Z 363.273,A -85,B 0,C 180,E1 -24089.026,E2 -24089.026} C_VEL
LIN {X 0,Y 150.239,Z 363.271,A -85,B 0,C 180,E1 -24092.722,E2 -24092.722} C_VEL
LIN {X 0,Y 150.348,Z 363.249,A -85,B 0,C 180,E1 -24099.211,E2 -24099.211} C_VEL
LIN {X 0,Y 150.367,Z 363.252,A -85,B 0,C 180,E1 -24103.715,E2 -24103.715} C_VEL
LIN {X 0,Y 150.652,Z 363.213,A -85,B 0,C 180,E1 -24109.247,E2 -24109.247} C_VEL
LIN {X 0,Y 150.739,Z 363.205,A -85,B 0,C 180,E1 -24111.961,E2 -24111.961} C_VEL
LIN {X 0,Y 151.217,Z 363.116,A -85,B 0,C 180,E1 -24120.001,E2 -24120.001} C_VEL
LIN {X 0,Y 150.743,Z 363.21,A -85,B 0,C 180,E1 -24128.042,E2 -24128.042} C_VEL
LIN {X 0,Y 150.607,Z 363.227,A -85,B 0,C 180,E1 -24131.492,E2 -24131.492} C_VEL
LIN {X 0,Y 150.35,Z 363.259,A -85,B 0,C 180,E1 -24136.289,E2 -24136.289} C_VEL
LIN {X 0,Y 150.371,Z 363.366,A -85,B 0,C 180,E1 -24139.098,E2 -24139.098} C_VEL
LIN {X 0,Y 150.452,Z 364.684,A -85,B 0,C 180,E1 -24144.862,E2 -24144.862} C_VEL
LIN {X 0,Y 150.51,Z 365.453,A -85,B 0,C 180,E1 -24147.838,E2 -24147.838} C_VEL
LIN {X 0,Y 150.717,Z 366.884,A -85,B 0,C 180,E1 -24152.929,E2 -24152.929} C_VEL
LIN {X 0,Y 150.808,Z 367.612,A -85,B 0,C 180,E1 -24155.017,E2 -24155.017} C_VEL
LIN {X 0,Y 151.976,Z 370.831,A -85,B 0,C 180,E1 -24156.029,E2 -24156.029} C_VEL
LIN {X 0,Y 154.193,Z 373.697,A -85,B 0,C 180,E1 -24157.551,E2 -24157.551} C_VEL
LIN {X 0,Y 155.919,Z 377.422,A -85,B 0,C 180,E1 -24158.903,E2 -24158.903} C_VEL
LIN {X 0,Y 157.102,Z 379.406,A -85,B 0,C 180,E1 -24159.711,E2 -24159.711} C_VEL
LIN {X 0,Y 160.757,Z 387.887,A -85,B 0,C 180,E1 -24162.661,E2 -24162.661} C_VEL
LIN {X 0,Y 163.001,Z 395.087,A -85,B 0,C 180,E1 -24164.888,E2 -24164.888} C_VEL
LIN {X 0,Y 164.712,Z 403.791,A -85,B 0,C 180,E1 -24167.394,E2 -24167.394} C_VEL
LIN {X 0,Y 165.598,Z 412.207,A -85,B 0,C 180,E1 -24169.813,E2 -24169.813} C_VEL
LIN {X 0,Y 165.791,Z 421.005,A -85,B 0,C 180,E1 -24172.46,E2 -24172.46} C_VEL
LIN {X 0,Y 165.327,Z 429.37,A -85,B 0,C 180,E1 -24175.187,E2 -24175.187} C_VEL
LIN {X 0,Y 164.627,Z 434.638,A -85,B 0,C 180,E1 -24177.023,E2 -24177.023} C_VEL
LIN {X 0,Y 162.618,Z 439.651,A -85,B 0,C 180,E1 -24178.761,E2 -24178.761} C_VEL
LIN {X 0,Y 159.847,Z 445.601,A -85,B 0,C 180,E1 -24181.077,E2 -24181.077} C_VEL
LIN {X 0,Y 157.417,Z 450.764,A -85,B 0,C 180,E1 -24183.484,E2 -24183.484} C_VEL
LIN {X 0,Y 155.22,Z 455.268,A -85,B 0,C 180,E1 -24185.952,E2 -24185.952} C_VEL
LIN {X 0,Y 152.374,Z 460.76,A -85,B 0,C 180,E1 -24189.762,E2 -24189.762} C_VEL
LIN {X 0,Y 150.148,Z 465.087,A -85,B 0,C 180,E1 -24193.69,E2 -24193.69} C_VEL
LIN {X 0,Y 149.17,Z 467.46,A -85,B 0,C 180,E1 -24196.375,E2 -24196.375} C_VEL
LIN {X 0,Y 148.406,Z 469.265,A -85,B 0,C 180,E1 -24199.081,E2 -24199.081} C_VEL
LIN {X 0,Y 147.687,Z 471.725,A -85,B 0,C 180,E1 -24204.539,E2 -24204.539} C_VEL
LIN {X 0,Y 147.628,Z 472.476,A -85,B 0,C 180,E1 -24208.729,E2 -24208.729} C_VEL
LIN {X 0,Y 147.572,Z 472.318,A -85,B 0,C 180,E1 -24212.73,E2 -24212.73} C_VEL
LIN {X 0,Y 147.638,Z 471.723,A -85,B 0,C 180,E1 -24215.463,E2 -24215.463} C_VEL
LIN {X 0,Y 148.406,Z 469.265,A -85,B 0,C 180,E1 -24220.919,E2 -24220.919} C_VEL
LIN {X 0,Y 149.643,Z 466.307,A -85,B 0,C 180,E1 -24224.97,E2 -24224.97} C_VEL
LIN {X 0,Y 151.56,Z 462.314,A -85,B 0,C 180,E1 -24228.941,E2 -24228.941} C_VEL
LIN {X 0,Y 154.183,Z 457.183,A -85,B 0,C 180,E1 -24232.796,E2 -24232.796} C_VEL
LIN {X 0,Y 156.907,Z 451.922,A -85,B 0,C 180,E1 -24235.894,E2 -24235.894} C_VEL
LIN {X 0,Y 159.844,Z 445.601,A -85,B 0,C 180,E1 -24238.924,E2 -24238.924} C_VEL
LIN {X 0,Y 162.574,Z 439.65,A -85,B 0,C 180,E1 -24241.249,E2 -24241.249} C_VEL
LIN {X 0,Y 164.629,Z 434.638,A -85,B 0,C 180,E1 -24242.976,E2 -24242.976} C_VEL
LIN {X 0,Y 165.635,Z 425.739,A -85,B 0,C 180,E1 -24246.017,E2 -24246.017} C_VEL
LIN {X 0,Y 165.827,Z 417.232,A -85,B 0,C 180,E1 -24248.68,E2 -24248.68} C_VEL
LIN {X 0,Y 165.308,Z 408.335,A -85,B 0,C 180,E1 -24251.295,E2 -24251.295} C_VEL
LIN {X 0,Y 163.991,Z 399.721,A -85,B 0,C 180,E1 -24253.797,E2 -24253.797} C_VEL
LIN {X 0,Y 161.831,Z 390.868,A -85,B 0,C 180,E1 -24256.414,E2 -24256.414} C_VEL
LIN {X 0,Y 158.652,Z 382.685,A -85,B 0,C 180,E1 -24259.115,E2 -24259.115} C_VEL
LIN {X 0,Y 156.487,Z 378.217,A -85,B 0,C 180,E1 -24260.729,E2 -24260.729} C_VEL
LIN {X 0,Y 154.42,Z 374.421,A -85,B 0,C 180,E1 -24262.232,E2 -24262.232} C_VEL
LIN {X 0,Y 153.915,Z 373.241,A -85,B 0,C 180,E1 -24262.652,E2 -24262.652} C_VEL
LIN {X 0,Y 153.398,Z 372.727,A -85,B 0,C 180,E1 -24262.982,E2 -24262.982} C_VEL
LIN {X 0,Y 149.501,Z 369.794,A -85,B 0,C 180,E1 -24265.468,E2 -24265.468} C_VEL
LIN {X 0,Y 144.01,Z 367.349,A -85,B 0,C 180,E1 -24269.069,E2 -24269.069} C_VEL
LIN {X 0,Y 143.504,Z 367.059,A -85,B 0,C 180,E1 -24269.933,E2 -24269.933} C_VEL
LIN {X 0,Y 143.416,Z 366.071,A -85,B 0,C 180,E1 -24273.828,E2 -24273.828} C_VEL
LIN {X 0,Y 143.374,Z 364.697,A -85,B 0,C 180,E1 -24279.931,E2 -24279.931} C_VEL
LIN {X 0,Y 143.297,Z 364.137,A -85,B 0,C 180,E1 -24282.885,E2 -24282.885} C_VEL
LIN {X 0,Y 143.595,Z 364.099,A -85,B 0,C 180,E1 -24288.709,E2 -24288.709} C_VEL
LIN {X 0,Y 143.662,Z 364.091,A -85,B 0,C 180,E1 -24291.559,E2 -24291.559} C_VEL
LIN {X 0,Y 144.176,Z 363.991,A -85,B 0,C 180,E1 -24299.998,E2 -24299.998} C_VEL
LIN {X 0,Y 143.66,Z 364.083,A -85,B 0,C 180,E1 -24308.438,E2 -24308.438} C_VEL
LIN {X 0,Y 143.547,Z 364.104,A -85,B 0,C 180,E1 -24311.711,E2 -24311.711} C_VEL
LIN {X 0,Y 143.304,Z 364.136,A -85,B 0,C 180,E1 -24317.111,E2 -24317.111} C_VEL
LIN {X 0,Y 143.274,Z 364.133,A -85,B 0,C 180,E1 -24321.251,E2 -24321.251} C_VEL
LIN {X 0,Y 143.187,Z 364.149,A -85,B 0,C 180,E1 -24327.934,E2 -24327.934} C_VEL
LIN {X 0,Y 143.151,Z 364.152,A -85,B 0,C 180,E1 -24330.517,E2 -24330.517} C_VEL
LIN {X 0,Y 144.056,Z 366.826,A -85,B 0,C 180,E1 -24331.527,E2 -24331.527} C_VEL
LIN {X 0,Y 146.385,Z 369.266,A -85,B 0,C 180,E1 -24333.442,E2 -24333.442} C_VEL
LIN {X 0,Y 146.979,Z 370.029,A -85,B 0,C 180,E1 -24333.932,E2 -24333.932} C_VEL
LIN {X 0,Y 148.648,Z 372.969,A -85,B 0,C 180,E1 -24335.391,E2 -24335.391} C_VEL
LIN {X 0,Y 150.188,Z 374.813,A -85,B 0,C 180,E1 -24336.523,E2 -24336.523} C_VEL
LIN {X 0,Y 151.769,Z 377.607,A -85,B 0,C 180,E1 -24337.859,E2 -24337.859} C_VEL
LIN {X 0,Y 152.597,Z 378.58,A -85,B 0,C 180,E1 -24338.469,E2 -24338.469} C_VEL
LIN {X 0,Y 157.117,Z 386.671,A -85,B 0,C 180,E1 -24342.14,E2 -24342.14} C_VEL
LIN {X 0,Y 161.114,Z 395.508,A -85,B 0,C 180,E1 -24345.738,E2 -24345.738} C_VEL
LIN {X 0,Y 164.433,Z 404.828,A -85,B 0,C 180,E1 -24349.335,E2 -24349.335} C_VEL
LIN {X 0,Y 166.737,Z 413.974,A -85,B 0,C 180,E1 -24352.796,E2 -24352.796} C_VEL
LIN {X 0,Y 168.14,Z 422.49,A -85,B 0,C 180,E1 -24356.12,E2 -24356.12} C_VEL
LIN {X 0,Y 169.322,Z 428.588,A -85,B 0,C 180,E1 -24358.747,E2 -24358.747} C_VEL
LIN {X 0,Y 171.851,Z 436.173,A -85,B 0,C 180,E1 -24362.608,E2 -24362.608} C_VEL
LIN {X 0,Y 175.53,Z 442.455,A -85,B 0,C 180,E1 -24366.398,E2 -24366.398} C_VEL
LIN {X 0,Y 179.79,Z 447.26,A -85,B 0,C 180,E1 -24369.741,E2 -24369.741} C_VEL
LIN {X 0,Y 186.142,Z 452.152,A -85,B 0,C 180,E1 -24373.731,E2 -24373.731} C_VEL
LIN {X 0,Y 194.168,Z 456.245,A -85,B 0,C 180,E1 -24377.757,E2 -24377.757} C_VEL
LIN {X 0,Y 199.721,Z 458.304,A -85,B 0,C 180,E1 -24380.154,E2 -24380.154} C_VEL
LIN {X 0,Y 205.581,Z 459.926,A -85,B 0,C 180,E1 -24382.469,E2 -24382.469} C_VEL
LIN {X 0,Y 211.725,Z 461.118,A -85,B 0,C 180,E1 -24384.747,E2 -24384.747} C_VEL
LIN {X 0,Y 218.133,Z 461.962,A -85,B 0,C 180,E1 -24387.152,E2 -24387.152} C_VEL
LIN {X 0,Y 220.598,Z 462.19,A -85,B 0,C 180,E1 -24388.174,E2 -24388.174} C_VEL
LIN {X 0,Y 224.309,Z 462.261,A -85,B 0,C 180,E1 -24390,E2 -24390} C_VEL
LIN {X 0,Y 220.611,Z 462.19,A -85,B 0,C 180,E1 -24391.826,E2 -24391.826} C_VEL
LIN {X 0,Y 215.8,Z 461.753,A -85,B 0,C 180,E1 -24393.735,E2 -24393.735} C_VEL
LIN {X 0,Y 210.351,Z 460.876,A -85,B 0,C 180,E1 -24395.753,E2 -24395.753} C_VEL
LIN {X 0,Y 204.663,Z 459.687,A -85,B 0,C 180,E1 -24397.895,E2 -24397.895} C_VEL
LIN {X 0,Y 198.914,Z 458.06,A -85,B 0,C 180,E1 -24400.175,E2 -24400.175} C_VEL
LIN {X 0,Y 188.957,Z 453.806,A -85,B 0,C 180,E1 -24404.757,E2 -24404.757} C_VEL
LIN {X 0,Y 183.427,Z 450.365,A -85,B 0,C 180,E1 -24407.85,E2 -24407.85} C_VEL
LIN {X 0,Y 177.318,Z 444.686,A -85,B 0,C 180,E1 -24412.106,E2 -24412.106} C_VEL
LIN {X 0,Y 173.247,Z 438.857,A -85,B 0,C 180,E1 -24415.838,E2 -24415.838} C_VEL
LIN {X 0,Y 170.596,Z 432.905,A -85,B 0,C 180,E1 -24419.129,E2 -24419.129} C_VEL
LIN {X 0,Y 168.558,Z 425.011,A -85,B 0,C 180,E1 -24422.822,E2 -24422.822} C_VEL
LIN {X 0,Y 167.313,Z 417.03,A -85,B 0,C 180,E1 -24426.02,E2 -24426.02} C_VEL
LIN {X 0,Y 165.725,Z 409.736,A -85,B 0,C 180,E1 -24428.813,E2 -24428.813} C_VEL
LIN {X 0,Y 163.566,Z 402.395,A -85,B 0,C 180,E1 -24431.616,E2 -24431.616} C_VEL
LIN {X 0,Y 160.733,Z 394.572,A -85,B 0,C 180,E1 -24434.636,E2 -24434.636} C_VEL
LIN {X 0,Y 156.428,Z 385.42,A -85,B 0,C 180,E1 -24438.435,E2 -24438.435} C_VEL
LIN {X 0,Y 152.593,Z 378.58,A -85,B 0,C 180,E1 -24441.533,E2 -24441.533} C_VEL
LIN {X 0,Y 150.28,Z 375.001,A -85,B 0,C 180,E1 -24443.399,E2 -24443.399} C_VEL
LIN {X 0,Y 149.27,Z 373.641,A -85,B 0,C 180,E1 -24444.157,E2 -24444.157} C_VEL
LIN {X 0,Y 147.286,Z 370.769,A -85,B 0,C 180,E1 -24445.758,E2 -24445.758} C_VEL
LIN {X 0,Y 146.547,Z 369.361,A -85,B 0,C 180,E1 -24446.444,E2 -24446.444} C_VEL
LIN {X 0,Y 144.14,Z 366.978,A -85,B 0,C 180,E1 -24448.391,E2 -24448.391} C_VEL
LIN {X 0,Y 143.205,Z 364.504,A -85,B 0,C 180,E1 -24449.393,E2 -24449.393} C_VEL
LIN {X 0,Y 143.131,Z 364.155,A -85,B 0,C 180,E1 -24449.58,E2 -24449.58} C_VEL
LIN {X 0,Y 143.152,Z 364.148,A -85,B 0,C 180,E1 -24453.78,E2 -24453.78} C_VEL
LIN {X 0,Y 143.305,Z 364.124,A -85,B 0,C 180,E1 -24459.924,E2 -24459.924} C_VEL
LIN {X 0,Y 143.369,Z 364.117,A -85,B 0,C 180,E1 -24465.814,E2 -24465.814} C_VEL
LIN {X 0,Y 143.594,Z 364.095,A -85,B 0,C 180,E1 -24468.712,E2 -24468.712} C_VEL
LIN {X 0,Y 143.66,Z 364.083,A -85,B 0,C 180,E1 -24471.562,E2 -24471.562} C_VEL
LIN {X 0,Y 144.176,Z 363.991,A -85,B 0,C 180,E1 -24480.002,E2 -24480.002} C_VEL
LIN {X 0,Y 143.662,Z 364.091,A -85,B 0,C 180,E1 -24488.441,E2 -24488.441} C_VEL
LIN {X 0,Y 143.549,Z 364.107,A -85,B 0,C 180,E1 -24491.714,E2 -24491.714} C_VEL
LIN {X 0,Y 143.297,Z 364.138,A -85,B 0,C 180,E1 -24497.115,E2 -24497.115} C_VEL
LIN {X 0,Y 143.386,Z 364.968,A -85,B 0,C 180,E1 -24501.366,E2 -24501.366} C_VEL
LIN {X 0,Y 143.473,Z 366.562,A -85,B 0,C 180,E1 -24508.149,E2 -24508.149} C_VEL
LIN {X 0,Y 143.589,Z 367.365,A -85,B 0,C 180,E1 -24510.723,E2 -24510.723} C_VEL
